# B&R Automation Studio project pneutrunk_plc (part 2)

#### regulator_FF_PI.c
```c
/*
 * regulator_FF_PI.c
 *
 * Academic License - for use in teaching, academic research, and meeting
 * course requirements at degree granting institutions only.  Not for
 * government, commercial, or other organizational use.
 *
 * Code generation for model "regulator_FF_PI".
 *
 * Model version              : 1.96
 * Simulink Coder version : 9.6 (R2021b) 14-May-2021
 * C source code generated on : Tue Apr  5 15:19:23 2022
 *
 * Target selection: bur_grt.tlc
 * Note: GRT includes extra infrastructure and instrumentation for prototyping
 * Embedded hardware selection: Intel->x86/Pentium
 * Code generation objectives: Unspecified
 * Validation result: Not run
 */

#include "regulator_FF_PI.h"
#include "regulator_FF_PI_private.h"

/* Forward declaration for local functions */
static real32_T regulator_FF_PI_norm(const real32_T x[4], struct FF_PID* inst);

/* Function for MATLAB Function: '<S5>/requested alfa 2 deltaz1' */
static real32_T regulator_FF_PI_norm(const real32_T x[4], struct FF_PID* inst)
{
  real32_T absxk;
  real32_T scale;
  real32_T t;
  real32_T y;
  scale = 1.29246971E-26F;
  absxk = fabsf(x[0]);
  if (absxk > 1.29246971E-26F) {
    y = 1.0F;
    scale = absxk;
  } else {
    t = absxk / 1.29246971E-26F;
    y = t * t;
  }

  absxk = fabsf(x[1]);
  if (absxk > scale) {
    t = scale / absxk;
    y = y * t * t + 1.0F;
    scale = absxk;
  } else {
    t = absxk / scale;
    y += t * t;
  }

  absxk = fabsf(x[2]);
  if (absxk > scale) {
    t = scale / absxk;
    y = y * t * t + 1.0F;
    scale = absxk;
  } else {
    t = absxk / scale;
    y += t * t;
  }

  absxk = fabsf(x[3]);
  if (absxk > scale) {
    t = scale / absxk;
    y = y * t * t + 1.0F;
    scale = absxk;
  } else {
    t = absxk / scale;
    y += t * t;
  }

  return scale * sqrtf(y);
}

/* Model step function */
void regulator_FF_PI_step(RT_MODEL_regulator_FF_PI_T *const regulator_FF_PI_M, struct FF_PID* inst)
{
  B_regulator_FF_PI_T *regulator_FF_PI_B = regulator_FF_PI_M->blockIO;
  DW_regulator_FF_PI_T *regulator_FF_PI_DW = regulator_FF_PI_M->dwork;
  real_T oblast_bodov[114];
  real_T Tz23[16];
  real_T Blue0_tmp[4];
  real_T Yellow0_tmp[4];
  real_T A1;
  real_T A2;
  real_T rtb_out;
  real_T tlaky_idx_0;
  real_T tlaky_idx_1;
  real_T tlaky_idx_2;
  real_T tmp;
  real_T tolerancia_bodov;
  real_T tolerancia_tlakov;
  int32_T Tz23_tmp;
  int32_T counter3;
  int32_T i;
  int32_T k;
  real32_T rtb_MultiportSwitch[114];
  real32_T rozdiel[95];
  real32_T vzd_bodov[76];
  real32_T AlphaY_0[16];
  real32_T HTransform[16];
  real32_T HTransform_tmp_1[16];
  real32_T Tz23_0[16];
  real32_T Blue0_tmp_0[4];
  real32_T Green0_tmp_tmp_0[4];
  real32_T Yellow0_tmp_0[4];
  real32_T Yellow0_tmp_1[4];
  real32_T AlphaX;
  real32_T AlphaY;
  real32_T akt_u_idx_2;
  real32_T akt_u_idx_3;
  real32_T akt_u_idx_4;
  real32_T rozdiel_tmp;
  real32_T vzd_bodov_tmp;
  int8_T Green0_tmp_tmp[4];
  int8_T HTransform_tmp[4];
  int8_T HTransform_tmp_0[4];

  /* S-Function (bur_in): '<Root>/Input1' */
  regulator_FF_PI_B->Input1 = inst->ref_alfa_x;

  /* S-Function (bur_in): '<Root>/Input2' */
  regulator_FF_PI_B->Input2 = inst->ref_alfa_y;

  /* S-Function (bur_in): '<Root>/Input3' */
  regulator_FF_PI_B->Input3 = inst->real_alfa_x;

  /* S-Function (bur_in): '<Root>/Input4' */
  regulator_FF_PI_B->Input4 = inst->real_alfa_y;

  /* MATLAB Function: '<S5>/requested alfa 2 deltaz1' incorporates:
   *  Constant: '<S5>/Constant1'
   */
  AlphaX = regulator_FF_PI_B->Input1 * 3.14159274F / 180.0F;
  AlphaY = -regulator_FF_PI_B->Input2 * 3.14159274F / 180.0F;
  Tz23[2] = 0.0;
  Tz23[6] = 0.0;
  Tz23[10] = 1.0;
  Tz23[14] = 57.5;
  akt_u_idx_2 = sinf(AlphaY);
  AlphaY = cosf(AlphaY);
  akt_u_idx_3 = sinf(AlphaX);
  AlphaX = cosf(AlphaX);
  AlphaY_0[0] = AlphaY;
  AlphaY_0[4] = 0.0F;
  AlphaY_0[8] = akt_u_idx_2;
  AlphaY_0[12] = 0.0F;
  AlphaY_0[2] = -akt_u_idx_2;
  AlphaY_0[6] = 0.0F;
  AlphaY_0[10] = AlphaY;
  AlphaY_0[14] = 0.0F;
  Tz23[0] = 1.0;
  Tz23[1] = 0.0;
  Tz23[3] = 0.0;
  HTransform_tmp_0[0] = 1;
  AlphaY_0[1] = 0.0F;
  AlphaY_0[3] = 0.0F;
  HTransform_tmp[0] = 0;
  Tz23[4] = 0.0;
  Tz23[5] = 1.0;
  Tz23[7] = 0.0;
  HTransform_tmp_0[1] = 0;
  AlphaY_0[5] = 1.0F;
  AlphaY_0[7] = 0.0F;
  HTransform_tmp[1] = 0;
  Tz23[8] = 0.0;
  Tz23[9] = 0.0;
  Tz23[11] = 0.0;
  HTransform_tmp_0[2] = 0;
  AlphaY_0[9] = 0.0F;
  AlphaY_0[11] = 0.0F;
  HTransform_tmp[2] = 0;
  Tz23[12] = 0.0;
  Tz23[13] = 0.0;
  Tz23[15] = 1.0;
  HTransform_tmp_0[3] = 0;
  AlphaY_0[13] = 0.0F;
  AlphaY_0[15] = 1.0F;
  HTransform_tmp[3] = 1;
  HTransform_tmp_1[1] = 0.0F;
  HTransform_tmp_1[5] = AlphaX;
  HTransform_tmp_1[9] = -akt_u_idx_3;
  HTransform_tmp_1[13] = 0.0F;
  HTransform_tmp_1[2] = 0.0F;
  HTransform_tmp_1[6] = akt_u_idx_3;
  HTransform_tmp_1[10] = AlphaX;
  HTransform_tmp_1[14] = 0.0F;
  for (i = 0; i < 4; i++) {
    for (k = 0; k < 4; k++) {
      counter3 = k << 2;
      Tz23_tmp = i + counter3;
      Tz23_0[Tz23_tmp] = 0.0F;
      Tz23_0[Tz23_tmp] += AlphaY_0[counter3] * (real32_T)Tz23[i];
      Tz23_0[Tz23_tmp] += AlphaY_0[counter3 + 1] * (real32_T)Tz23[i + 4];
      Tz23_0[Tz23_tmp] += AlphaY_0[counter3 + 2] * (real32_T)Tz23[i + 8];
      Tz23_0[Tz23_tmp] += AlphaY_0[counter3 + 3] * (real32_T)Tz23[i + 12];
    }

    counter3 = i << 2;
    HTransform_tmp_1[counter3] = HTransform_tmp_0[i];
    HTransform_tmp_1[counter3 + 3] = HTransform_tmp[i];
  }

  Green0_tmp_tmp[0] = 85;
  Green0_tmp_tmp[1] = 0;
  Green0_tmp_tmp[2] = 0;
  Green0_tmp_tmp[3] = 1;
  Yellow0_tmp[0] = -42.5;
  Yellow0_tmp[1] = 73.612159321677282;
  Yellow0_tmp[2] = 0.0;
  Yellow0_tmp[3] = 1.0;
  Blue0_tmp[0] = -42.5;
  Blue0_tmp[1] = -73.612159321677282;
  Blue0_tmp[2] = 0.0;
  Blue0_tmp[3] = 1.0;
  for (i = 0; i < 4; i++) {
    for (k = 0; k < 4; k++) {
      counter3 = k << 2;
      Tz23_tmp = i + counter3;
      AlphaY_0[Tz23_tmp] = 0.0F;
      AlphaY_0[Tz23_tmp] += HTransform_tmp_1[counter3] * Tz23_0[i];
      AlphaY_0[Tz23_tmp] += HTransform_tmp_1[counter3 + 1] * Tz23_0[i + 4];
      AlphaY_0[Tz23_tmp] += HTransform_tmp_1[counter3 + 2] * Tz23_0[i + 8];
      AlphaY_0[Tz23_tmp] += HTransform_tmp_1[counter3 + 3] * Tz23_0[i + 12];
    }

    akt_u_idx_2 = 0.0F;
    akt_u_idx_3 = 0.0F;
    akt_u_idx_4 = 0.0F;
    for (k = 0; k < 4; k++) {
      counter3 = k << 2;
      Tz23_tmp = i + counter3;
      HTransform[Tz23_tmp] = 0.0F;
      HTransform[Tz23_tmp] += (real32_T)Tz23[counter3] * AlphaY_0[i];
      HTransform[Tz23_tmp] += (real32_T)Tz23[counter3 + 1] * AlphaY_0[i + 4];
      HTransform[Tz23_tmp] += (real32_T)Tz23[counter3 + 2] * AlphaY_0[i + 8];
      HTransform[Tz23_tmp] += (real32_T)Tz23[counter3 + 3] * AlphaY_0[i + 12];
      akt_u_idx_2 += HTransform[Tz23_tmp] * (real32_T)Green0_tmp_tmp[k];
      akt_u_idx_3 += HTransform[Tz23_tmp] * (real32_T)Yellow0_tmp[k];
      akt_u_idx_4 += HTransform[Tz23_tmp] * (real32_T)Blue0_tmp[k];
    }

    Green0_tmp_tmp_0[i] = (real32_T)Green0_tmp_tmp[i] - akt_u_idx_2;
    Yellow0_tmp_0[i] = (real32_T)Yellow0_tmp[i] - akt_u_idx_3;
    Blue0_tmp_0[i] = (real32_T)Blue0_tmp[i] - akt_u_idx_4;
  }

  AlphaX = regulator_FF_PI_B->Input3 * 3.14159274F / 180.0F;
  AlphaY = -regulator_FF_PI_B->Input4 * 3.14159274F / 180.0F;
  akt_u_idx_2 = sinf(AlphaY);
  AlphaY = cosf(AlphaY);
  akt_u_idx_3 = sinf(AlphaX);
  AlphaX = cosf(AlphaX);
  AlphaY_0[0] = AlphaY;
  AlphaY_0[4] = 0.0F;
  AlphaY_0[8] = akt_u_idx_2;
  AlphaY_0[12] = 0.0F;
  AlphaY_0[2] = -akt_u_idx_2;
  AlphaY_0[6] = 0.0F;
  AlphaY_0[10] = AlphaY;
  AlphaY_0[14] = 0.0F;
  AlphaY_0[1] = 0.0F;
  AlphaY_0[3] = 0.0F;
  AlphaY_0[5] = 1.0F;
  AlphaY_0[7] = 0.0F;
  AlphaY_0[9] = 0.0F;
  AlphaY_0[11] = 0.0F;
  AlphaY_0[13] = 0.0F;
  AlphaY_0[15] = 1.0F;
  HTransform_tmp_1[1] = 0.0F;
  HTransform_tmp_1[5] = AlphaX;
  HTransform_tmp_1[9] = -akt_u_idx_3;
  HTransform_tmp_1[13] = 0.0F;
  HTransform_tmp_1[2] = 0.0F;
  HTransform_tmp_1[6] = akt_u_idx_3;
  HTransform_tmp_1[10] = AlphaX;
  HTransform_tmp_1[14] = 0.0F;
  for (i = 0; i < 4; i++) {
    for (k = 0; k < 4; k++) {
      counter3 = k << 2;
      Tz23_tmp = i + counter3;
      Tz23_0[Tz23_tmp] = 0.0F;
      Tz23_0[Tz23_tmp] += AlphaY_0[counter3] * (real32_T)Tz23[i];
      Tz23_0[Tz23_tmp] += AlphaY_0[counter3 + 1] * (real32_T)Tz23[i + 4];
      Tz23_0[Tz23_tmp] += AlphaY_0[counter3 + 2] * (real32_T)Tz23[i + 8];
      Tz23_0[Tz23_tmp] += AlphaY_0[counter3 + 3] * (real32_T)Tz23[i + 12];
    }

    counter3 = i << 2;
    HTransform_tmp_1[counter3] = HTransform_tmp_0[i];
    HTransform_tmp_1[counter3 + 3] = HTransform_tmp[i];
  }

  Yellow0_tmp[0] = -42.5;
  Yellow0_tmp[1] = 73.612159321677282;
  Yellow0_tmp[2] = 0.0;
  Yellow0_tmp[3] = 1.0;
  Blue0_tmp[0] = -42.5;
  Blue0_tmp[1] = -73.612159321677282;
  Blue0_tmp[2] = 0.0;
  Blue0_tmp[3] = 1.0;
  for (i = 0; i < 4; i++) {
    for (k = 0; k < 4; k++) {
      counter3 = k << 2;
      Tz23_tmp = i + counter3;
      AlphaY_0[Tz23_tmp] = 0.0F;
      AlphaY_0[Tz23_tmp] += HTransform_tmp_1[counter3] * Tz23_0[i];
      AlphaY_0[Tz23_tmp] += HTransform_tmp_1[counter3 + 1] * Tz23_0[i + 4];
      AlphaY_0[Tz23_tmp] += HTransform_tmp_1[counter3 + 2] * Tz23_0[i + 8];
      AlphaY_0[Tz23_tmp] += HTransform_tmp_1[counter3 + 3] * Tz23_0[i + 12];
    }

    akt_u_idx_2 = 0.0F;
    for (k = 0; k < 4; k++) {
      counter3 = k << 2;
      Tz23_tmp = i + counter3;
      HTransform[Tz23_tmp] = 0.0F;
      HTransform[Tz23_tmp] += (real32_T)Tz23[counter3] * AlphaY_0[i];
      HTransform[Tz23_tmp] += (real32_T)Tz23[counter3 + 1] * AlphaY_0[i + 4];
      HTransform[Tz23_tmp] += (real32_T)Tz23[counter3 + 2] * AlphaY_0[i + 8];
      HTransform[Tz23_tmp] += (real32_T)Tz23[counter3 + 3] * AlphaY_0[i + 12];
      akt_u_idx_2 += HTransform[Tz23_tmp] * (real32_T)Yellow0_tmp[k];
    }

    Yellow0_tmp_1[i] = (real32_T)Yellow0_tmp[i] - akt_u_idx_2;
  }

  /* Sum: '<S2>/Sum' incorporates:
   *  Constant: '<S11>/cylinder height'
   *  Constant: '<S9>/cylinder height'
   *  Gain: '<S5>/Gain'
   *  Gain: '<S5>/Gain3'
   *  MATLAB Function: '<S5>/requested alfa 2 deltaz1'
   *  Sum: '<S11>/Sum'
   *  Sum: '<S9>/Sum'
   */
  A2 = (0.001F * regulator_FF_PI_norm(Yellow0_tmp_1, inst) - 0.115) - (0.001F *
    regulator_FF_PI_norm(Yellow0_tmp_0, inst) - 0.115);

  /* S-Function (bur_in): '<Root>/Input11' */
  regulator_FF_PI_B->Input11 = inst->P_parameter;

  /* S-Function (bur_in): '<Root>/Input5' */
  regulator_FF_PI_B->Input5 = inst->reset_PID_blue;

  /* DiscreteIntegrator: '<S143>/Integrator' */
  if ((regulator_FF_PI_B->Input5 <= 0.0F) &&
      (regulator_FF_PI_DW->Integrator_PrevResetState == 1)) {
    regulator_FF_PI_DW->Integrator_DSTATE = 0.0;
  }

  /* S-Function (bur_in): '<Root>/Input13' */
  regulator_FF_PI_B->Input13 = inst->D_parameter;

  /* DiscreteIntegrator: '<S138>/Filter' */
  if ((regulator_FF_PI_B->Input5 <= 0.0F) &&
      (regulator_FF_PI_DW->Filter_PrevResetState == 1)) {
    regulator_FF_PI_DW->Filter_DSTATE = 0.0;
  }

  /* S-Function (bur_in): '<Root>/Input14' */
  regulator_FF_PI_B->Input14 = inst->N_parameter;

  /* Product: '<S146>/NProd Out' incorporates:
   *  DiscreteIntegrator: '<S138>/Filter'
   *  Product: '<S137>/DProd Out'
   *  Sum: '<S138>/SumD'
   */
  A1 = (A2 * regulator_FF_PI_B->Input13 - regulator_FF_PI_DW->Filter_DSTATE) *
    regulator_FF_PI_B->Input14;

  /* S-Function (bur_in): '<Root>/Input8' */
  regulator_FF_PI_B->Input8 = inst->tlak1;

  /* S-Function (bur_in): '<Root>/Input9' */
  regulator_FF_PI_B->Input9 = inst->tlak2;

  /* S-Function (bur_in): '<Root>/Input10' */
  regulator_FF_PI_B->Input10 = inst->tlak3;

  /* MATLAB Function: '<S1>/prepinac' */
  rtb_out = 1.0;
  if ((regulator_FF_PI_B->Input1 < 0.0F) && (regulator_FF_PI_B->Input2 > 0.0F))
  {
    rtb_out = 2.0;
  }

  if ((regulator_FF_PI_B->Input1 > 0.0F) && (regulator_FF_PI_B->Input2 < 0.0F))
  {
    rtb_out = 3.0;
  }

  if ((regulator_FF_PI_B->Input1 <= 0.0F) && (regulator_FF_PI_B->Input2 <= 0.0F))
  {
    rtb_out = 4.0;
  }

  /* End of MATLAB Function: '<S1>/prepinac' */

  /* MultiPortSwitch: '<S1>/Multiport Switch' incorporates:
   *  Constant: '<S1>/Constant'
   *  Constant: '<S1>/Constant1'
   *  Constant: '<S1>/Constant2'
   *  Constant: '<S1>/Constant3'
   */
  switch ((int32_T)rtb_out) {
   case 1:
    for (i = 0; i < 114; i++) {
      rtb_MultiportSwitch[i] = regulator_FF_PI_ConstP.Constant_Value_m[i];
    }
    break;

   case 2:
    for (i = 0; i < 114; i++) {
      rtb_MultiportSwitch[i] = regulator_FF_PI_ConstP.Constant1_Value_b[i];
    }
    break;

   case 3:
    for (i = 0; i < 114; i++) {
      rtb_MultiportSwitch[i] = regulator_FF_PI_ConstP.Constant3_Value[i];
    }
    break;

   default:
    for (i = 0; i < 114; i++) {
      rtb_MultiportSwitch[i] = regulator_FF_PI_ConstP.Constant2_Value[i];
    }
    break;
  }

  /* End of MultiPortSwitch: '<S1>/Multiport Switch' */

  /* MATLAB Function: '<S1>/ff' incorporates:
   *  MultiPortSwitch: '<S1>/Multiport Switch'
   */
  akt_u_idx_2 = regulator_FF_PI_B->Input8;
  akt_u_idx_3 = regulator_FF_PI_B->Input9;
  akt_u_idx_4 = regulator_FF_PI_B->Input10;
  tolerancia_bodov = 2.0;
  tolerancia_tlakov = 2.0;
  counter3 = 0;
  tlaky_idx_0 = 0.0;
  tlaky_idx_1 = 0.0;
  tlaky_idx_2 = 0.0;
  for (k = 0; k < 19; k++) {
    rozdiel[k] = rtb_MultiportSwitch[k] - regulator_FF_PI_B->Input1;
    rozdiel[k + 19] = rtb_MultiportSwitch[k + 19] - regulator_FF_PI_B->Input2;
    AlphaX = rtb_MultiportSwitch[k + 38];
    rozdiel[k + 38] = AlphaX;
    AlphaY = rtb_MultiportSwitch[k + 57];
    rozdiel[k + 57] = AlphaY;
    rozdiel_tmp = rtb_MultiportSwitch[k + 76];
    rozdiel[k + 76] = rozdiel_tmp;
    vzd_bodov_tmp = rozdiel[k + 19];
    vzd_bodov[k] = sqrtf(vzd_bodov_tmp * vzd_bodov_tmp + rozdiel[k] * rozdiel[k]);
    vzd_bodov[k + 19] = AlphaX;
    vzd_bodov[k + 38] = AlphaY;
    vzd_bodov[k + 57] = rozdiel_tmp;
  }

  for (i = 0; i < 114; i++) {
    oblast_bodov[i] = 0.0;
  }

  rtb_out = 0.0;
  if (regulator_FF_PI_B->Input8 <= 2.0F) {
    akt_u_idx_2 = 2.0F;
  }

  if (regulator_FF_PI_B->Input9 <= 2.0F) {
    akt_u_idx_3 = 2.0F;
  }

  if (regulator_FF_PI_B->Input10 <= 2.0F) {
    akt_u_idx_4 = 2.0F;
  }

  int32_T exitg1;
  do {
    exitg1 = 0;
    for (k = 0; k < 19; k++) {
      if ((vzd_bodov[k] <= tolerancia_bodov) && (fabsf(((akt_u_idx_2 +
              akt_u_idx_3) + akt_u_idx_4) - rtb_MultiportSwitch[k + 95]) <=
           tolerancia_tlakov)) {
        rtb_out++;
        for (i = 0; i < 6; i++) {
          oblast_bodov[((int32_T)rtb_out + 19 * i) - 1] = rtb_MultiportSwitch[19
            * i + k];
        }

        rozdiel_tmp = (real32_T)oblast_bodov[(int32_T)rtb_out - 1] -
          regulator_FF_PI_B->Input1;
        vzd_bodov_tmp = (real32_T)oblast_bodov[(int32_T)rtb_out + 18] -
          regulator_FF_PI_B->Input2;
        rozdiel_tmp = sqrtf(rozdiel_tmp * rozdiel_tmp + vzd_bodov_tmp *
                            vzd_bodov_tmp);
        if (rozdiel_tmp <= 0.5F) {
          if (counter3 == 0) {
            counter3 = 1;
            tlaky_idx_0 = oblast_bodov[(int32_T)rtb_out + 37];
            tlaky_idx_1 = oblast_bodov[(int32_T)rtb_out + 56];
            tlaky_idx_2 = oblast_bodov[(int32_T)rtb_out + 75];
          } else {
            AlphaX = (real32_T)oblast_bodov[(int32_T)(rtb_out - 1.0) - 1] -
              regulator_FF_PI_B->Input1;
            AlphaY = (real32_T)oblast_bodov[(int32_T)(rtb_out - 1.0) + 18] -
              regulator_FF_PI_B->Input2;
            if (rozdiel_tmp < sqrtf(AlphaX * AlphaX + AlphaY * AlphaY)) {
              tlaky_idx_0 = oblast_bodov[(int32_T)rtb_out + 37];
              tlaky_idx_1 = oblast_bodov[(int32_T)rtb_out + 56];
              tlaky_idx_2 = oblast_bodov[(int32_T)rtb_out + 75];
            }
          }
        }
      }
    }

    if (rtb_out == 0.0) {
      tolerancia_bodov++;
      tolerancia_tlakov++;
    } else {
      exitg1 = 1;
    }
  } while (exitg1 == 0);

  if (counter3 == 0) {
    tolerancia_bodov = oblast_bodov[38];
    for (counter3 = 2; counter3 <= (int32_T)rtb_out; counter3++) {
      tolerancia_bodov += oblast_bodov[counter3 + 37];
    }

    tolerancia_tlakov = oblast_bodov[57];
    for (counter3 = 2; counter3 <= (int32_T)rtb_out; counter3++) {
      tolerancia_tlakov += oblast_bodov[counter3 + 56];
    }

    tlaky_idx_2 = oblast_bodov[76];
    for (counter3 = 2; counter3 <= (int32_T)rtb_out; counter3++) {
      tlaky_idx_2 += oblast_bodov[counter3 + 75];
    }

    tlaky_idx_0 = tolerancia_bodov / (real_T)(int32_T)rtb_out;
    tlaky_idx_1 = tolerancia_tlakov / (real_T)(int32_T)rtb_out;
    tlaky_idx_2 /= (real_T)(int32_T)rtb_out;
  }

  /* Switch: '<Root>/Switch2' incorporates:
   *  DiscreteIntegrator: '<S143>/Integrator'
   *  Product: '<S148>/PProd Out'
   *  Sum: '<S152>/Sum'
   */
  if (regulator_FF_PI_B->Input5 > 0.0F) {
    tmp = (A2 * regulator_FF_PI_B->Input11 +
           regulator_FF_PI_DW->Integrator_DSTATE) + A1;
  } else {
    tmp = 0.0;
  }

  /* End of Switch: '<Root>/Switch2' */

  /* Sum: '<Root>/Sum' incorporates:
   *  MATLAB Function: '<S1>/ff'
   */
  regulator_FF_PI_B->Sum = (real32_T)(tmp + tlaky_idx_0);

  /* S-Function (bur_out): '<Root>/Output1' */
  inst->Blue_tab = regulator_FF_PI_B->Sum;

  /* MATLAB Function: '<S5>/requested alfa 2 deltaz1' */
  for (i = 0; i < 4; i++) {
    Yellow0_tmp_0[i] = (real32_T)Green0_tmp_tmp[i] - (HTransform[i] * 85.0F +
      HTransform[i + 12]);
  }

  /* Sum: '<S2>/Sum2' incorporates:
   *  Constant: '<S12>/cylinder height'
   *  Constant: '<S14>/cylinder height'
   *  Gain: '<S5>/Gain1'
   *  Gain: '<S5>/Gain4'
   *  MATLAB Function: '<S5>/requested alfa 2 deltaz1'
   *  Sum: '<S12>/Sum'
   *  Sum: '<S14>/Sum'
   */
  tolerancia_tlakov = (0.001F * regulator_FF_PI_norm(Yellow0_tmp_0, inst) - 0.115) -
    (0.001F * regulator_FF_PI_norm(Green0_tmp_tmp_0, inst) - 0.115);

  /* S-Function (bur_in): '<Root>/Input7' */
  regulator_FF_PI_B->Input7 = inst->reset_PID_green;

  /* DiscreteIntegrator: '<S95>/Integrator' */
  if ((regulator_FF_PI_B->Input7 <= 0.0F) &&
      (regulator_FF_PI_DW->Integrator_PrevResetState_l == 1)) {
    regulator_FF_PI_DW->Integrator_DSTATE_o = 0.0;
  }

  /* DiscreteIntegrator: '<S90>/Filter' */
  if ((regulator_FF_PI_B->Input7 <= 0.0F) &&
      (regulator_FF_PI_DW->Filter_PrevResetState_e == 1)) {
    regulator_FF_PI_DW->Filter_DSTATE_f = 0.0;
  }

  /* Product: '<S98>/NProd Out' incorporates:
   *  DiscreteIntegrator: '<S90>/Filter'
   *  Product: '<S89>/DProd Out'
   *  Sum: '<S90>/SumD'
   */
  rtb_out = (tolerancia_tlakov * regulator_FF_PI_B->Input13 -
             regulator_FF_PI_DW->Filter_DSTATE_f) * regulator_FF_PI_B->Input14;

  /* Switch: '<Root>/Switch' incorporates:
   *  DiscreteIntegrator: '<S95>/Integrator'
   *  Product: '<S100>/PProd Out'
   *  Sum: '<S104>/Sum'
   */
  if (regulator_FF_PI_B->Input7 > 0.0F) {
    tmp = (tolerancia_tlakov * regulator_FF_PI_B->Input11 +
           regulator_FF_PI_DW->Integrator_DSTATE_o) + rtb_out;
  } else {
    tmp = 0.0;
  }

  /* End of Switch: '<Root>/Switch' */

  /* Sum: '<Root>/Sum2' incorporates:
   *  MATLAB Function: '<S1>/ff'
   */
  regulator_FF_PI_B->Sum2 = (real32_T)(tmp + tlaky_idx_2);

  /* S-Function (bur_out): '<Root>/Output2' */
  inst->Yellow_tab = regulator_FF_PI_B->Sum2;

  /* MATLAB Function: '<S5>/requested alfa 2 deltaz1' */
  for (i = 0; i < 4; i++) {
    Green0_tmp_tmp_0[i] = (real32_T)Blue0_tmp[i] - ((HTransform[i + 4] *
      -73.6121597F + HTransform[i] * -42.5F) + HTransform[i + 12]);
  }

  /* Sum: '<S2>/Sum1' incorporates:
   *  Constant: '<S10>/cylinder height'
   *  Constant: '<S13>/cylinder height'
   *  Gain: '<S5>/Gain2'
   *  Gain: '<S5>/Gain5'
   *  MATLAB Function: '<S5>/requested alfa 2 deltaz1'
   *  Sum: '<S10>/Sum'
   *  Sum: '<S13>/Sum'
   */
  tlaky_idx_2 = (0.001F * regulator_FF_PI_norm(Green0_tmp_tmp_0, inst) - 0.115) -
    (0.001F * regulator_FF_PI_norm(Blue0_tmp_0, inst) - 0.115);

  /* S-Function (bur_in): '<Root>/Input6' */
  regulator_FF_PI_B->Input6 = inst->reset_PID_yellow;

  /* DiscreteIntegrator: '<S47>/Integrator' */
  if ((regulator_FF_PI_B->Input6 <= 0.0F) &&
      (regulator_FF_PI_DW->Integrator_PrevResetState_e == 1)) {
    regulator_FF_PI_DW->Integrator_DSTATE_i = 0.0;
  }

  /* DiscreteIntegrator: '<S42>/Filter' */
  if ((regulator_FF_PI_B->Input6 <= 0.0F) &&
      (regulator_FF_PI_DW->Filter_PrevResetState_h == 1)) {
    regulator_FF_PI_DW->Filter_DSTATE_a = 0.0;
  }

  /* Product: '<S50>/NProd Out' incorporates:
   *  DiscreteIntegrator: '<S42>/Filter'
   *  Product: '<S41>/DProd Out'
   *  Sum: '<S42>/SumD'
   */
  tolerancia_bodov = (tlaky_idx_2 * regulator_FF_PI_B->Input13 -
                      regulator_FF_PI_DW->Filter_DSTATE_a) *
    regulator_FF_PI_B->Input14;

  /* Switch: '<Root>/Switch1' incorporates:
   *  DiscreteIntegrator: '<S47>/Integrator'
   *  Product: '<S52>/PProd Out'
   *  Sum: '<S56>/Sum'
   */
  if (regulator_FF_PI_B->Input6 > 0.0F) {
    tmp = (tlaky_idx_2 * regulator_FF_PI_B->Input11 +
           regulator_FF_PI_DW->Integrator_DSTATE_i) + tolerancia_bodov;
  } else {
    tmp = 0.0;
  }

  /* End of Switch: '<Root>/Switch1' */

  /* Sum: '<Root>/Sum1' incorporates:
   *  MATLAB Function: '<S1>/ff'
   */
  regulator_FF_PI_B->Sum1 = (real32_T)(tmp + tlaky_idx_1);

  /* S-Function (bur_out): '<Root>/Output4' */
  inst->Green_tab = regulator_FF_PI_B->Sum1;

  /* S-Function (bur_in): '<Root>/Input12' */
  regulator_FF_PI_B->Input12 = inst->I_parameter;

  /* Product: '<S44>/IProd Out' */
  tlaky_idx_0 = tlaky_idx_2 * regulator_FF_PI_B->Input12;

  /* Product: '<S92>/IProd Out' */
  tolerancia_tlakov *= regulator_FF_PI_B->Input12;

  /* Product: '<S140>/IProd Out' */
  A2 *= regulator_FF_PI_B->Input12;

  /* Update for DiscreteIntegrator: '<S143>/Integrator' */
  regulator_FF_PI_DW->Integrator_DSTATE += 0.002 * A2;
  if (regulator_FF_PI_B->Input5 > 0.0F) {
    regulator_FF_PI_DW->Integrator_PrevResetState = 1;
  } else if (regulator_FF_PI_B->Input5 < 0.0F) {
    regulator_FF_PI_DW->Integrator_PrevResetState = -1;
  } else if (regulator_FF_PI_B->Input5 == 0.0F) {
    regulator_FF_PI_DW->Integrator_PrevResetState = 0;
  } else {
    regulator_FF_PI_DW->Integrator_PrevResetState = 2;
  }

  /* End of Update for DiscreteIntegrator: '<S143>/Integrator' */

  /* Update for DiscreteIntegrator: '<S138>/Filter' */
  regulator_FF_PI_DW->Filter_DSTATE += 0.002 * A1;
  if (regulator_FF_PI_B->Input5 > 0.0F) {
    regulator_FF_PI_DW->Filter_PrevResetState = 1;
  } else if (regulator_FF_PI_B->Input5 < 0.0F) {
    regulator_FF_PI_DW->Filter_PrevResetState = -1;
  } else if (regulator_FF_PI_B->Input5 == 0.0F) {
    regulator_FF_PI_DW->Filter_PrevResetState = 0;
  } else {
    regulator_FF_PI_DW->Filter_PrevResetState = 2;
  }

  /* End of Update for DiscreteIntegrator: '<S138>/Filter' */

  /* Update for DiscreteIntegrator: '<S95>/Integrator' */
  regulator_FF_PI_DW->Integrator_DSTATE_o += 0.002 * tolerancia_tlakov;
  if (regulator_FF_PI_B->Input7 > 0.0F) {
    regulator_FF_PI_DW->Integrator_PrevResetState_l = 1;
  } else if (regulator_FF_PI_B->Input7 < 0.0F) {
    regulator_FF_PI_DW->Integrator_PrevResetState_l = -1;
  } else if (regulator_FF_PI_B->Input7 == 0.0F) {
    regulator_FF_PI_DW->Integrator_PrevResetState_l = 0;
  } else {
    regulator_FF_PI_DW->Integrator_PrevResetState_l = 2;
  }

  /* End of Update for DiscreteIntegrator: '<S95>/Integrator' */

  /* Update for DiscreteIntegrator: '<S90>/Filter' */
  regulator_FF_PI_DW->Filter_DSTATE_f += 0.002 * rtb_out;
  if (regulator_FF_PI_B->Input7 > 0.0F) {
    regulator_FF_PI_DW->Filter_PrevResetState_e = 1;
  } else if (regulator_FF_PI_B->Input7 < 0.0F) {
    regulator_FF_PI_DW->Filter_PrevResetState_e = -1;
  } else if (regulator_FF_PI_B->Input7 == 0.0F) {
    regulator_FF_PI_DW->Filter_PrevResetState_e = 0;
  } else {
    regulator_FF_PI_DW->Filter_PrevResetState_e = 2;
  }

  /* End of Update for DiscreteIntegrator: '<S90>/Filter' */

  /* Update for DiscreteIntegrator: '<S47>/Integrator' */
  regulator_FF_PI_DW->Integrator_DSTATE_i += 0.002 * tlaky_idx_0;
  if (regulator_FF_PI_B->Input6 > 0.0F) {
    regulator_FF_PI_DW->Integrator_PrevResetState_e = 1;
  } else if (regulator_FF_PI_B->Input6 < 0.0F) {
    regulator_FF_PI_DW->Integrator_PrevResetState_e = -1;
  } else if (regulator_FF_PI_B->Input6 == 0.0F) {
    regulator_FF_PI_DW->Integrator_PrevResetState_e = 0;
  } else {
    regulator_FF_PI_DW->Integrator_PrevResetState_e = 2;
  }

  /* End of Update for DiscreteIntegrator: '<S47>/Integrator' */

  /* Update for DiscreteIntegrator: '<S42>/Filter' */
  regulator_FF_PI_DW->Filter_DSTATE_a += 0.002 * tolerancia_bodov;
  if (regulator_FF_PI_B->Input6 > 0.0F) {
    regulator_FF_PI_DW->Filter_PrevResetState_h = 1;
  } else if (regulator_FF_PI_B->Input6 < 0.0F) {
    regulator_FF_PI_DW->Filter_PrevResetState_h = -1;
  } else if (regulator_FF_PI_B->Input6 == 0.0F) {
    regulator_FF_PI_DW->Filter_PrevResetState_h = 0;
  } else {
    regulator_FF_PI_DW->Filter_PrevResetState_h = 2;
  }

  /* End of Update for DiscreteIntegrator: '<S42>/Filter' */
}

/* Model initialize function */
void regulator_FF_PI_initialize(RT_MODEL_regulator_FF_PI_T *const
  regulator_FF_PI_M, struct FF_PID* inst)
{
  DW_regulator_FF_PI_T *regulator_FF_PI_DW = regulator_FF_PI_M->dwork;

  /* InitializeConditions for DiscreteIntegrator: '<S143>/Integrator' */
  regulator_FF_PI_DW->Integrator_DSTATE = 0.0;
  regulator_FF_PI_DW->Integrator_PrevResetState = 2;

  /* InitializeConditions for DiscreteIntegrator: '<S138>/Filter' */
  regulator_FF_PI_DW->Filter_DSTATE = 0.0;
  regulator_FF_PI_DW->Filter_PrevResetState = 2;

  /* InitializeConditions for DiscreteIntegrator: '<S95>/Integrator' */
  regulator_FF_PI_DW->Integrator_DSTATE_o = 0.0;
  regulator_FF_PI_DW->Integrator_PrevResetState_l = 2;

  /* InitializeConditions for DiscreteIntegrator: '<S90>/Filter' */
  regulator_FF_PI_DW->Filter_DSTATE_f = 0.0;
  regulator_FF_PI_DW->Filter_PrevResetState_e = 2;

  /* InitializeConditions for DiscreteIntegrator: '<S47>/Integrator' */
  regulator_FF_PI_DW->Integrator_DSTATE_i = 0.0;
  regulator_FF_PI_DW->Integrator_PrevResetState_e = 2;

  /* InitializeConditions for DiscreteIntegrator: '<S42>/Filter' */
  regulator_FF_PI_DW->Filter_DSTATE_a = 0.0;
  regulator_FF_PI_DW->Filter_PrevResetState_h = 2;
}

/* Model terminate function */
void regulator_FF_PI_terminate(RT_MODEL_regulator_FF_PI_T * regulator_FF_PI_M, struct FF_PID* inst)
{}

/* Model data allocation function */
void regulator_FF_PI_initializeMemory(RT_MODEL_regulator_FF_PI_T* const regulator_FF_PI_M, struct FF_PID * inst)
{  /* states (dwork) */
  {
  }

  {
    B_regulator_FF_PI_T *regulator_FF_PI_B = regulator_FF_PI_M->blockIO;
    DW_regulator_FF_PI_T *regulator_FF_PI_DW = regulator_FF_PI_M->dwork;

    /* block I/O */
    {
      regulator_FF_PI_B->Input1 = 0.0F;
      regulator_FF_PI_B->Input2 = 0.0F;
      regulator_FF_PI_B->Input3 = 0.0F;
      regulator_FF_PI_B->Input4 = 0.0F;
      regulator_FF_PI_B->Input11 = 0.0F;
      regulator_FF_PI_B->Input5 = 0.0F;
      regulator_FF_PI_B->Input13 = 0.0F;
      regulator_FF_PI_B->Input14 = 0.0F;
      regulator_FF_PI_B->Input8 = 0.0F;
      regulator_FF_PI_B->Input9 = 0.0F;
      regulator_FF_PI_B->Input10 = 0.0F;
      regulator_FF_PI_B->Sum = 0.0F;
      regulator_FF_PI_B->Input7 = 0.0F;
      regulator_FF_PI_B->Sum2 = 0.0F;
      regulator_FF_PI_B->Input6 = 0.0F;
      regulator_FF_PI_B->Sum1 = 0.0F;
      regulator_FF_PI_B->Input12 = 0.0F;
    }

    /* states (dwork) */
    (void) memset((void *)regulator_FF_PI_DW, 0,
                  sizeof(DW_regulator_FF_PI_T));
    regulator_FF_PI_DW->Integrator_DSTATE = 0.0;
    regulator_FF_PI_DW->Filter_DSTATE = 0.0;
    regulator_FF_PI_DW->Integrator_DSTATE_o = 0.0;
    regulator_FF_PI_DW->Filter_DSTATE_f = 0.0;
    regulator_FF_PI_DW->Integrator_DSTATE_i = 0.0;
    regulator_FF_PI_DW->Filter_DSTATE_a = 0.0;
  }

}
```

#### regulator_nelin_P.c
```c
/*
 * regulator_nelin_P.c
 *
 * Academic License - for use in teaching, academic research, and meeting
 * course requirements at degree granting institutions only.  Not for
 * government, commercial, or other organizational use.
 *
 * Code generation for model "regulator_nelin_P".
 *
 * Model version              : 1.10
 * Simulink Coder version : 9.6 (R2021b) 14-May-2021
 * C source code generated on : Fri Jul 29 10:48:17 2022
 *
 * Target selection: bur_grt.tlc
 * Note: GRT includes extra infrastructure and instrumentation for prototyping
 * Embedded hardware selection: Intel->x86/Pentium
 * Code generation objectives: Unspecified
 * Validation result: Not run
 */

#include "regulator_nelin_P.h"
#include "regulator_nelin_P_private.h"

/* Forward declaration for local functions */
static real32_T regulator_nelin_P_norm(const real32_T x[4], struct nonL_P* inst);

/* Function for MATLAB Function: '<S1>/requested alfa 2 deltaz1' */
static real32_T regulator_nelin_P_norm(const real32_T x[4], struct nonL_P* inst)
{
  real32_T absxk;
  real32_T scale;
  real32_T t;
  real32_T y;
  scale = 1.29246971E-26F;
  absxk = fabsf(x[0]);
  if (absxk > 1.29246971E-26F) {
    y = 1.0F;
    scale = absxk;
  } else {
    t = absxk / 1.29246971E-26F;
    y = t * t;
  }

  absxk = fabsf(x[1]);
  if (absxk > scale) {
    t = scale / absxk;
    y = y * t * t + 1.0F;
    scale = absxk;
  } else {
    t = absxk / scale;
    y += t * t;
  }

  absxk = fabsf(x[2]);
  if (absxk > scale) {
    t = scale / absxk;
    y = y * t * t + 1.0F;
    scale = absxk;
  } else {
    t = absxk / scale;
    y += t * t;
  }

  absxk = fabsf(x[3]);
  if (absxk > scale) {
    t = scale / absxk;
    y = y * t * t + 1.0F;
    scale = absxk;
  } else {
    t = absxk / scale;
    y += t * t;
  }

  return scale * sqrtf(y);
}

/* Model step function */
void regulator_nelin_P_step(RT_MODEL_regulator_nelin_P_T *const
  regulator_nelin_P_M, struct nonL_P* inst)
{
  B_regulator_nelin_P_T *regulator_nelin_P_B = regulator_nelin_P_M->blockIO;
  real_T Tz23[16];
  real_T Blue0_tmp[4];
  real_T Yellow0_tmp[4];
  int32_T Tz23_tmp;
  int32_T Tz23_tmp_tmp;
  int32_T i;
  int32_T i_0;
  real32_T AlphaY_0[16];
  real32_T HTransform[16];
  real32_T HTransform_tmp_3[16];
  real32_T Tz23_0[16];
  real32_T Blue0_tmp_0[4];
  real32_T Green0_tmp_tmp_0[4];
  real32_T Yellow0_tmp_0[4];
  real32_T Yellow0_tmp_1[4];
  real32_T AlphaX;
  real32_T AlphaY;
  real32_T HTransform_tmp;
  real32_T HTransform_tmp_0;
  int8_T Green0_tmp_tmp[4];
  int8_T HTransform_tmp_1[4];
  int8_T HTransform_tmp_2[4];

  /* S-Function (bur_in): '<Root>/Input1' */
  regulator_nelin_P_B->Input1 = inst->ref_alfa_x;

  /* S-Function (bur_in): '<Root>/Input2' */
  regulator_nelin_P_B->Input2 = inst->ref_alfa_y;

  /* S-Function (bur_in): '<Root>/Input3' */
  regulator_nelin_P_B->Input3 = inst->real_alfa_x;

  /* S-Function (bur_in): '<Root>/Input4' */
  regulator_nelin_P_B->Input4 = inst->real_alfa_y;

  /* MATLAB Function: '<S1>/requested alfa 2 deltaz1' incorporates:
   *  Constant: '<S1>/Constant1'
   */
  AlphaX = regulator_nelin_P_B->Input1 * 3.14159274F / 180.0F;
  AlphaY = -regulator_nelin_P_B->Input2 * 3.14159274F / 180.0F;
  Tz23[2] = 0.0;
  Tz23[6] = 0.0;
  Tz23[10] = 1.0;
  Tz23[14] = 57.5;
  HTransform_tmp = sinf(AlphaY);
  AlphaY = cosf(AlphaY);
  HTransform_tmp_0 = sinf(AlphaX);
  AlphaX = cosf(AlphaX);
  AlphaY_0[0] = AlphaY;
  AlphaY_0[4] = 0.0F;
  AlphaY_0[8] = HTransform_tmp;
  AlphaY_0[12] = 0.0F;
  AlphaY_0[2] = -HTransform_tmp;
  AlphaY_0[6] = 0.0F;
  AlphaY_0[10] = AlphaY;
  AlphaY_0[14] = 0.0F;
  Tz23[0] = 1.0;
  Tz23[1] = 0.0;
  Tz23[3] = 0.0;
  HTransform_tmp_2[0] = 1;
  AlphaY_0[1] = 0.0F;
  AlphaY_0[3] = 0.0F;
  HTransform_tmp_1[0] = 0;
  Tz23[4] = 0.0;
  Tz23[5] = 1.0;
  Tz23[7] = 0.0;
  HTransform_tmp_2[1] = 0;
  AlphaY_0[5] = 1.0F;
  AlphaY_0[7] = 0.0F;
  HTransform_tmp_1[1] = 0;
  Tz23[8] = 0.0;
  Tz23[9] = 0.0;
  Tz23[11] = 0.0;
  HTransform_tmp_2[2] = 0;
  AlphaY_0[9] = 0.0F;
  AlphaY_0[11] = 0.0F;
  HTransform_tmp_1[2] = 0;
  Tz23[12] = 0.0;
  Tz23[13] = 0.0;
  Tz23[15] = 1.0;
  HTransform_tmp_2[3] = 0;
  AlphaY_0[13] = 0.0F;
  AlphaY_0[15] = 1.0F;
  HTransform_tmp_1[3] = 1;
  HTransform_tmp_3[1] = 0.0F;
  HTransform_tmp_3[5] = AlphaX;
  HTransform_tmp_3[9] = -HTransform_tmp_0;
  HTransform_tmp_3[13] = 0.0F;
  HTransform_tmp_3[2] = 0.0F;
  HTransform_tmp_3[6] = HTransform_tmp_0;
  HTransform_tmp_3[10] = AlphaX;
  HTransform_tmp_3[14] = 0.0F;
  for (i = 0; i < 4; i++) {
    for (i_0 = 0; i_0 < 4; i_0++) {
      Tz23_tmp_tmp = i_0 << 2;
      Tz23_tmp = i + Tz23_tmp_tmp;
      Tz23_0[Tz23_tmp] = 0.0F;
      Tz23_0[Tz23_tmp] += AlphaY_0[Tz23_tmp_tmp] * (real32_T)Tz23[i];
      Tz23_0[Tz23_tmp] += AlphaY_0[Tz23_tmp_tmp + 1] * (real32_T)Tz23[i + 4];
      Tz23_0[Tz23_tmp] += AlphaY_0[Tz23_tmp_tmp + 2] * (real32_T)Tz23[i + 8];
      Tz23_0[Tz23_tmp] += AlphaY_0[Tz23_tmp_tmp + 3] * (real32_T)Tz23[i + 12];
    }

    Tz23_tmp_tmp = i << 2;
    HTransform_tmp_3[Tz23_tmp_tmp] = HTransform_tmp_2[i];
    HTransform_tmp_3[Tz23_tmp_tmp + 3] = HTransform_tmp_1[i];
  }

  Green0_tmp_tmp[0] = 85;
  Green0_tmp_tmp[1] = 0;
  Green0_tmp_tmp[2] = 0;
  Green0_tmp_tmp[3] = 1;
  Yellow0_tmp[0] = -42.5;
  Yellow0_tmp[1] = 73.612159321677282;
  Yellow0_tmp[2] = 0.0;
  Yellow0_tmp[3] = 1.0;
  Blue0_tmp[0] = -42.5;
  Blue0_tmp[1] = -73.612159321677282;
  Blue0_tmp[2] = 0.0;
  Blue0_tmp[3] = 1.0;
  for (i = 0; i < 4; i++) {
    for (i_0 = 0; i_0 < 4; i_0++) {
      Tz23_tmp_tmp = i_0 << 2;
      Tz23_tmp = i + Tz23_tmp_tmp;
      AlphaY_0[Tz23_tmp] = 0.0F;
      AlphaY_0[Tz23_tmp] += HTransform_tmp_3[Tz23_tmp_tmp] * Tz23_0[i];
      AlphaY_0[Tz23_tmp] += HTransform_tmp_3[Tz23_tmp_tmp + 1] * Tz23_0[i + 4];
      AlphaY_0[Tz23_tmp] += HTransform_tmp_3[Tz23_tmp_tmp + 2] * Tz23_0[i + 8];
      AlphaY_0[Tz23_tmp] += HTransform_tmp_3[Tz23_tmp_tmp + 3] * Tz23_0[i + 12];
    }

    AlphaX = 0.0F;
    AlphaY = 0.0F;
    HTransform_tmp = 0.0F;
    for (i_0 = 0; i_0 < 4; i_0++) {
      Tz23_tmp_tmp = i_0 << 2;
      Tz23_tmp = i + Tz23_tmp_tmp;
      HTransform[Tz23_tmp] = 0.0F;
      HTransform[Tz23_tmp] += (real32_T)Tz23[Tz23_tmp_tmp] * AlphaY_0[i];
      HTransform[Tz23_tmp] += (real32_T)Tz23[Tz23_tmp_tmp + 1] * AlphaY_0[i + 4];
      HTransform[Tz23_tmp] += (real32_T)Tz23[Tz23_tmp_tmp + 2] * AlphaY_0[i + 8];
      HTransform[Tz23_tmp] += (real32_T)Tz23[Tz23_tmp_tmp + 3] * AlphaY_0[i + 12];
      AlphaX += HTransform[Tz23_tmp] * (real32_T)Green0_tmp_tmp[i_0];
      AlphaY += HTransform[Tz23_tmp] * (real32_T)Yellow0_tmp[i_0];
      HTransform_tmp += HTransform[Tz23_tmp] * (real32_T)Blue0_tmp[i_0];
    }

    Green0_tmp_tmp_0[i] = (real32_T)Green0_tmp_tmp[i] - AlphaX;
    Yellow0_tmp_0[i] = (real32_T)Yellow0_tmp[i] - AlphaY;
    Blue0_tmp_0[i] = (real32_T)Blue0_tmp[i] - HTransform_tmp;
  }

  AlphaX = regulator_nelin_P_B->Input3 * 3.14159274F / 180.0F;
  AlphaY = -regulator_nelin_P_B->Input4 * 3.14159274F / 180.0F;
  HTransform_tmp = sinf(AlphaY);
  AlphaY = cosf(AlphaY);
  HTransform_tmp_0 = sinf(AlphaX);
  AlphaX = cosf(AlphaX);
  AlphaY_0[0] = AlphaY;
  AlphaY_0[4] = 0.0F;
  AlphaY_0[8] = HTransform_tmp;
  AlphaY_0[12] = 0.0F;
  AlphaY_0[2] = -HTransform_tmp;
  AlphaY_0[6] = 0.0F;
  AlphaY_0[10] = AlphaY;
  AlphaY_0[14] = 0.0F;
  AlphaY_0[1] = 0.0F;
  AlphaY_0[3] = 0.0F;
  AlphaY_0[5] = 1.0F;
  AlphaY_0[7] = 0.0F;
  AlphaY_0[9] = 0.0F;
  AlphaY_0[11] = 0.0F;
  AlphaY_0[13] = 0.0F;
  AlphaY_0[15] = 1.0F;
  HTransform_tmp_3[1] = 0.0F;
  HTransform_tmp_3[5] = AlphaX;
  HTransform_tmp_3[9] = -HTransform_tmp_0;
  HTransform_tmp_3[13] = 0.0F;
  HTransform_tmp_3[2] = 0.0F;
  HTransform_tmp_3[6] = HTransform_tmp_0;
  HTransform_tmp_3[10] = AlphaX;
  HTransform_tmp_3[14] = 0.0F;
  for (i = 0; i < 4; i++) {
    for (i_0 = 0; i_0 < 4; i_0++) {
      Tz23_tmp_tmp = i_0 << 2;
      Tz23_tmp = i + Tz23_tmp_tmp;
      Tz23_0[Tz23_tmp] = 0.0F;
      Tz23_0[Tz23_tmp] += AlphaY_0[Tz23_tmp_tmp] * (real32_T)Tz23[i];
      Tz23_0[Tz23_tmp] += AlphaY_0[Tz23_tmp_tmp + 1] * (real32_T)Tz23[i + 4];
      Tz23_0[Tz23_tmp] += AlphaY_0[Tz23_tmp_tmp + 2] * (real32_T)Tz23[i + 8];
      Tz23_0[Tz23_tmp] += AlphaY_0[Tz23_tmp_tmp + 3] * (real32_T)Tz23[i + 12];
    }

    Tz23_tmp_tmp = i << 2;
    HTransform_tmp_3[Tz23_tmp_tmp] = HTransform_tmp_2[i];
    HTransform_tmp_3[Tz23_tmp_tmp + 3] = HTransform_tmp_1[i];
  }

  Yellow0_tmp[0] = -42.5;
  Yellow0_tmp[1] = 73.612159321677282;
  Yellow0_tmp[2] = 0.0;
  Yellow0_tmp[3] = 1.0;
  Blue0_tmp[0] = -42.5;
  Blue0_tmp[1] = -73.612159321677282;
  Blue0_tmp[2] = 0.0;
  Blue0_tmp[3] = 1.0;
  for (i = 0; i < 4; i++) {
    for (i_0 = 0; i_0 < 4; i_0++) {
      Tz23_tmp_tmp = i_0 << 2;
      Tz23_tmp = i + Tz23_tmp_tmp;
      AlphaY_0[Tz23_tmp] = 0.0F;
      AlphaY_0[Tz23_tmp] += HTransform_tmp_3[Tz23_tmp_tmp] * Tz23_0[i];
      AlphaY_0[Tz23_tmp] += HTransform_tmp_3[Tz23_tmp_tmp + 1] * Tz23_0[i + 4];
      AlphaY_0[Tz23_tmp] += HTransform_tmp_3[Tz23_tmp_tmp + 2] * Tz23_0[i + 8];
      AlphaY_0[Tz23_tmp] += HTransform_tmp_3[Tz23_tmp_tmp + 3] * Tz23_0[i + 12];
    }

    AlphaX = 0.0F;
    for (i_0 = 0; i_0 < 4; i_0++) {
      Tz23_tmp_tmp = i_0 << 2;
      Tz23_tmp = i + Tz23_tmp_tmp;
      HTransform[Tz23_tmp] = 0.0F;
      HTransform[Tz23_tmp] += (real32_T)Tz23[Tz23_tmp_tmp] * AlphaY_0[i];
      HTransform[Tz23_tmp] += (real32_T)Tz23[Tz23_tmp_tmp + 1] * AlphaY_0[i + 4];
      HTransform[Tz23_tmp] += (real32_T)Tz23[Tz23_tmp_tmp + 2] * AlphaY_0[i + 8];
      HTransform[Tz23_tmp] += (real32_T)Tz23[Tz23_tmp_tmp + 3] * AlphaY_0[i + 12];
      AlphaX += HTransform[Tz23_tmp] * (real32_T)Yellow0_tmp[i_0];
    }

    Yellow0_tmp_1[i] = (real32_T)Yellow0_tmp[i] - AlphaX;
  }

  /* Gain: '<Root>/Gain7' incorporates:
   *  Constant: '<S3>/cylinder height'
   *  Constant: '<S5>/cylinder height'
   *  Gain: '<Root>/Gain3'
   *  Gain: '<Root>/Gain5'
   *  Gain: '<S1>/Gain'
   *  Gain: '<S1>/Gain3'
   *  MATLAB Function: '<Root>/MATLAB Function'
   *  MATLAB Function: '<S1>/requested alfa 2 deltaz1'
   *  Sum: '<S3>/Sum'
   *  Sum: '<S5>/Sum'
   */
  regulator_nelin_P_B->Gain7 = (real32_T)(pow(2.71828182845904, (0.001F *
    regulator_nelin_P_norm(Yellow0_tmp_0, inst) - 0.115) * 1000.0 * 0.1528) * 0.03078
    - pow(2.71828182845904, (0.001F * regulator_nelin_P_norm(Yellow0_tmp_1, inst) -
    0.115) * 1000.0 * 0.1528) * 0.03078);

  /* S-Function (bur_out): '<Root>/Output1' */
  inst->Blue_tab = regulator_nelin_P_B->Gain7;

  /* MATLAB Function: '<S1>/requested alfa 2 deltaz1' */
  for (i = 0; i < 4; i++) {
    Yellow0_tmp_0[i] = (real32_T)Blue0_tmp[i] - ((HTransform[i + 4] *
      -73.6121597F + HTransform[i] * -42.5F) + HTransform[i + 12]);
  }

  /* Gain: '<Root>/Gain9' incorporates:
   *  Constant: '<S6>/cylinder height'
   *  Constant: '<S8>/cylinder height'
   *  Gain: '<Root>/Gain2'
   *  Gain: '<Root>/Gain6'
   *  Gain: '<S1>/Gain2'
   *  Gain: '<S1>/Gain5'
   *  MATLAB Function: '<Root>/MATLAB Function'
   *  MATLAB Function: '<S1>/requested alfa 2 deltaz1'
   *  Sum: '<S6>/Sum'
   *  Sum: '<S8>/Sum'
   */
  regulator_nelin_P_B->Gain9 = (real32_T)(pow(2.71828182845904, (0.001F *
    regulator_nelin_P_norm(Blue0_tmp_0, inst) - 0.115) * 1000.0 * 0.1528) * 0.03078 -
    pow(2.71828182845904, (0.001F * regulator_nelin_P_norm(Yellow0_tmp_0, inst) -
    0.115) * 1000.0 * 0.1528) * 0.03078);

  /* S-Function (bur_out): '<Root>/Output2' */
  inst->Yellow_tab = regulator_nelin_P_B->Gain9;

  /* MATLAB Function: '<S1>/requested alfa 2 deltaz1' */
  for (i = 0; i < 4; i++) {
    Blue0_tmp_0[i] = (real32_T)Green0_tmp_tmp[i] - (HTransform[i] * 85.0F +
      HTransform[i + 12]);
  }

  /* Gain: '<Root>/Gain8' incorporates:
   *  Constant: '<S4>/cylinder height'
   *  Constant: '<S7>/cylinder height'
   *  Gain: '<Root>/Gain1'
   *  Gain: '<Root>/Gain4'
   *  Gain: '<S1>/Gain1'
   *  Gain: '<S1>/Gain4'
   *  MATLAB Function: '<Root>/MATLAB Function'
   *  MATLAB Function: '<S1>/requested alfa 2 deltaz1'
   *  Sum: '<S4>/Sum'
   *  Sum: '<S7>/Sum'
   */
  regulator_nelin_P_B->Gain8 = (real32_T)(pow(2.71828182845904, (0.001F *
    regulator_nelin_P_norm(Green0_tmp_tmp_0, inst) - 0.115) * 1000.0 * 0.1528) *
    0.03078 - pow(2.71828182845904, (0.001F * regulator_nelin_P_norm(Blue0_tmp_0, inst)
    - 0.115) * 1000.0 * 0.1528) * 0.03078);

  /* S-Function (bur_out): '<Root>/Output4' */
  inst->Green_tab = regulator_nelin_P_B->Gain8;
}

/* Model initialize function */
void regulator_nelin_P_initialize(RT_MODEL_regulator_nelin_P_T *const
  regulator_nelin_P_M, struct nonL_P* inst)
{
  UNUSED_PARAMETER(regulator_nelin_P_M);
}

/* Model terminate function */
void regulator_nelin_P_terminate(RT_MODEL_regulator_nelin_P_T
  * regulator_nelin_P_M, struct nonL_P* inst)
{}

/* Model data allocation function */
void regulator_nelin_P_initializeMemory(RT_MODEL_regulator_nelin_P_T* const regulator_nelin_P_M, struct nonL_P * inst)
{
  /* block I/O */
  {
  }

  {
    B_regulator_nelin_P_T *regulator_nelin_P_B = regulator_nelin_P_M->blockIO;

    /* block I/O */
    {
      regulator_nelin_P_B->Input1 = 0.0F;
      regulator_nelin_P_B->Input2 = 0.0F;
      regulator_nelin_P_B->Input3 = 0.0F;
      regulator_nelin_P_B->Input4 = 0.0F;
      regulator_nelin_P_B->Gain7 = 0.0F;
      regulator_nelin_P_B->Gain9 = 0.0F;
      regulator_nelin_P_B->Gain8 = 0.0F;
    }
  }

}
```

### Program Logical/Source/Program (IEC)

#### Variables.var
```iecst
VAR
	TON_0 : TON;
	TON_1 : TON;
	TON_2 : TON;
	TON_3 : TON;
	TON_4 : TON;
	i : INT;
END_VAR
```

#### Cyclic.st
```iecst
PROGRAM _CYCLIC

	TON_0(IN := automatika.casovac, PT := INT_TO_TIME(automatika.cas));
	TON_1(IN := automatika.casovac_uchopenie, PT := T#4s);
	//TON_2(IN := automatika.trajectoryStart, PT := automatika.trajectoryTime);
	//TON_4(IN := automatika.trajectoryStart2, PT := automatika.trajectoryTime2);
	//TON_3(IN := automatika.novyCyklusStart, PT := automatika.novyCyklus);

	CASE global_step OF

		0:	// caka kym spravi uvodne odmeranie referencii....v controlleri ak je krok 4, vtedy prechadza global_step = 1
			(*
			automatika.y_desired[0]	:= 0;
			automatika.y_desired[1]	:= 0;
			automatika.y_desired[2]	:= 0;
			automatika.y_desired[3]	:= 0;
			automatika.y_desired[4]	:= 0;
			automatika.y_desired[5]	:= 0;
			automatika.y_desired[6]	:= 0;

			automatika.x_desired[0]	:= 0;
			automatika.x_desired[1]	:= 0;
			automatika.x_desired[2]	:= 0;
			automatika.x_desired[3]	:= 0;
			automatika.x_desired[4]	:= 0;
			automatika.x_desired[5]	:= 0;
			automatika.x_desired[6]	:= 0;
			*)
			automatika.linear		:= 23;
			FOR i:=0 TO 6 BY 1 DO
				automatika.I_konstanta[i]	:= 5;
			END_FOR
			automatika.automatic	:= FALSE;
			(*
			IF automatika.step_color = 1 OR automatika.step_color = 2 THEN
				global_step				:= 999;
			END_IF
			*)
			modul;

		999:
			IF automatika.step_color = 1 OR automatika.step_color = 2 THEN
				automatika.loptickyVzasobniku	:= TRUE;
			ELSE
				automatika.loptickyVzasobniku	:= FALSE;
			END_IF

			IF automatika.loptickyVzasobniku = TRUE OR global_step_udp = 1 THEN
				automatika.effector		:= FALSE;
			//	global_step_udp			:= 0;
				global_step				:= 1;
				automatika.automatic	:= FALSE;
				I_ON					:= FALSE;
			END_IF
			FOR i:=0 TO 6 BY 1 DO
				automatika.I_konstanta[i]	:= 0;
			END_FOR

		1:
			automatika.cas			:= 1000;
			automatika.casovac		:= TRUE;
			I_ON					:= TRUE;
			global_step				:= 100;

		100:
			IF TON_0.Q = TRUE THEN
				automatika.casovac	:= FALSE;
				IF global_step_udp = 1 THEN
					global_step				:= 11;
				ELSE
					automatika.cas			:= 1000;
					automatika.casovac		:= TRUE;
					global_step				:= 2;
				END_IF
			END_IF

		2:
			IF TON_0.Q=TRUE THEN
				automatika.casovac		:= FALSE;
				//automatika.ball_up		:= TRUE;
				global_step				:= 3;
			//	automatika.ball_piston	:= FALSE;
			END_IF

		3:	// pohyb pre uchopenie gulicky
			//automatika.casovac_uchopenie	:= TRUE;
			IF(automatika.step_color = 1)THEN
				automatika.box := 1;
				automatika.loptickyVzasobniku := TRUE;
			ELSIF(automatika.step_color = 2)THEN
				automatika.box	:= 2;
				automatika.loptickyVzasobniku := TRUE;
			ELSIF(automatika.step_color = 3)THEN
				automatika.loptickyVzasobniku := FALSE;
				automatika.box := 3;
			END_IF

			automatika.casovac			:= TRUE;
			automatika.cas				:= 5000;
			automatika.effector			:= FALSE;
			automatika.linear			:= 23;
			global_step					:= 4;
			FOR i:=0 TO 6 BY 1 DO
				automatika.I_konstanta[i]	:= 30;
			END_FOR
		4:
			// Pohyb ku levitujucej lopte

			automatika.y_desired[0]	:= TIME_TO_INT(TON_0.ET)*(-7)/((automatika.cas));
			automatika.y_desired[1]	:= TIME_TO_INT(TON_0.ET)*(6)/((automatika.cas));
			automatika.y_desired[2]	:= TIME_TO_INT(TON_0.ET)*(-10)/((automatika.cas));
			automatika.y_desired[3]	:= TIME_TO_INT(TON_0.ET)*(-10)/((automatika.cas));
			automatika.y_desired[4]	:= TIME_TO_INT(TON_0.ET)*(-8)/((automatika.cas));
			automatika.y_desired[5]	:= TIME_TO_INT(TON_0.ET)*(-5)/((automatika.cas));
			automatika.y_desired[6]	:= TIME_TO_INT(TON_0.ET)*(-5)/((automatika.cas));//-10

			automatika.x_desired[0]	:= TIME_TO_INT(TON_0.ET)*5/((automatika.cas));
			automatika.x_desired[1]	:= TIME_TO_INT(TON_0.ET)*4/((automatika.cas));
			automatika.x_desired[2]	:= TIME_TO_INT(TON_0.ET)*5/((automatika.cas));
			automatika.x_desired[3]	:= TIME_TO_INT(TON_0.ET)*5/((automatika.cas));
			automatika.x_desired[4]	:= TIME_TO_INT(TON_0.ET)*5/((automatika.cas));
			automatika.x_desired[5]	:= TIME_TO_INT(TON_0.ET)*1/((automatika.cas));
			automatika.x_desired[6]	:= 0;// TIME_TO_INT(TON_0.ET)*2/((automatika.cas));

			//automatika.linear		:= TIME_TO_INT(TON_2.ET)*30/(TIME_TO_INT(automatika.trajectoryTime));

			IF TON_0.Q=TRUE THEN
				automatika.casovac			:= FALSE;
				automatika.casovac_uchopenie:= TRUE;
				global_step					:= 55;
				FOR i:=0 TO 6 BY 1 DO
					automatika.x_desired_previous[i]	:= automatika.x_desired[i];
					automatika.y_desired_previous[i]	:= automatika.y_desired[i];
					automatika.I_konstanta[i]			:= 20;
				END_FOR
			END_IF

		55:
			IF TON_1.Q = TRUE THEN
				automatika.levitacia			:= TRUE;
				automatika.linear				:= 30;
				automatika.casovac_uchopenie	:= FALSE;
				global_step						:= 555;
			END_IF

		555:
			automatika.cas						:= 1000;
			automatika.casovac					:= TRUE;
			global_step							:= 5;

		5:	// uchopenie
			IF TON_0.Q = TRUE THEN
				automatika.casovac				:= FALSE;
				automatika.effector				:= TRUE;
				global_step						:= 6;
			END_IF

		6:
			automatika.casovac_uchopenie		:= TRUE;
			global_step							:= 7;
			automatika.linear					:= 23;

		7:
			IF TON_1.Q = TRUE THEN
				automatika.casovac_uchopenie	:= FALSE;
				global_step						:= 8;
				automatika.levitacia			:= FALSE;
				automatika.ball_piston			:= TRUE;
				automatika.cas					:= 4500;
				automatika.casovac				:= TRUE;
				FOR i:=0 TO 6 BY 1 DO
					automatika.I_konstanta[i]	:= 50;
				END_FOR
			END_IF

		8:
			IF(automatika.box = 1) THEN
				// prenesenie objektu
				automatika.y_desired[0]	:= (automatika.y_desired_previous[0]*(automatika.cas - TIME_TO_INT(TON_0.ET))/automatika.cas) + TIME_TO_INT(TON_0.ET)*(7)/((automatika.cas));
				automatika.y_desired[1]	:= (automatika.y_desired_previous[1]*(automatika.cas - TIME_TO_INT(TON_0.ET))/automatika.cas) +  TIME_TO_INT(TON_0.ET)*(0)/((automatika.cas));	// 5000ms
				automatika.y_desired[2]	:= (automatika.y_desired_previous[2]*(automatika.cas - TIME_TO_INT(TON_0.ET))/automatika.cas) +  TIME_TO_INT(TON_0.ET)*(10)/((automatika.cas));
				automatika.y_desired[3]	:= (automatika.y_desired_previous[3]*(automatika.cas - TIME_TO_INT(TON_0.ET))/automatika.cas) +  TIME_TO_INT(TON_0.ET)*(0)/((automatika.cas));
				automatika.y_desired[4]	:= (automatika.y_desired_previous[4]*(automatika.cas - TIME_TO_INT(TON_0.ET))/automatika.cas) +  TIME_TO_INT(TON_0.ET)*(8)/((automatika.cas));
				automatika.y_desired[5]	:= (automatika.y_desired_previous[5]*(automatika.cas - TIME_TO_INT(TON_0.ET))/automatika.cas) +  TIME_TO_INT(TON_0.ET)*(5)/((automatika.cas));
				automatika.y_desired[6]	:= (automatika.y_desired_previous[6]*(automatika.cas - TIME_TO_INT(TON_0.ET))/automatika.cas) +  TIME_TO_INT(TON_0.ET)*(10)/((automatika.cas));

				automatika.x_desired[0]	:= (automatika.x_desired_previous[0]*(automatika.cas - TIME_TO_INT(TON_0.ET))/automatika.cas) +  TIME_TO_INT(TON_0.ET)*(2)/((automatika.cas));
				automatika.x_desired[1]	:= (automatika.x_desired_previous[1]*(automatika.cas - TIME_TO_INT(TON_0.ET))/automatika.cas) +  TIME_TO_INT(TON_0.ET)*(-2)/((automatika.cas));
				automatika.x_desired[2]	:= (automatika.x_desired_previous[2]*(automatika.cas - TIME_TO_INT(TON_0.ET))/automatika.cas) +  TIME_TO_INT(TON_0.ET)*(-2)/((automatika.cas));
				automatika.x_desired[3]	:= (automatika.x_desired_previous[3]*(automatika.cas - TIME_TO_INT(TON_0.ET))/automatika.cas) +  TIME_TO_INT(TON_0.ET)*(-2)/((automatika.cas));
				automatika.x_desired[4]	:= (automatika.x_desired_previous[4]*(automatika.cas - TIME_TO_INT(TON_0.ET))/automatika.cas) +  TIME_TO_INT(TON_0.ET)*(-5)/((automatika.cas));
				automatika.x_desired[5]	:= (automatika.x_desired_previous[5]*(automatika.cas - TIME_TO_INT(TON_0.ET))/automatika.cas) +  TIME_TO_INT(TON_0.ET)*(-5)/((automatika.cas));
				automatika.x_desired[6]	:= TIME_TO_INT(TON_0.ET)*(-5)/((automatika.cas));

				automatika.linear		:= TIME_TO_INT(TON_0.ET)*30/((automatika.cas));
			ELSIF(automatika.box = 2) THEN
				// prenesenie objektu
				automatika.y_desired[0]	:= (automatika.y_desired_previous[0]*(automatika.cas - TIME_TO_INT(TON_0.ET))/automatika.cas) + TIME_TO_INT(TON_0.ET)*(7)/((automatika.cas));
				automatika.y_desired[1]	:= (automatika.y_desired_previous[1]*(automatika.cas - TIME_TO_INT(TON_0.ET))/automatika.cas) + TIME_TO_INT(TON_0.ET)*(2)/((automatika.cas));	// 5000ms
				automatika.y_desired[2]	:= (automatika.y_desired_previous[2]*(automatika.cas - TIME_TO_INT(TON_0.ET))/automatika.cas) + TIME_TO_INT(TON_0.ET)*(10)/((automatika.cas));
				automatika.y_desired[3]	:= (automatika.y_desired_previous[3]*(automatika.cas - TIME_TO_INT(TON_0.ET))/automatika.cas) + TIME_TO_INT(TON_0.ET)*(0)/((automatika.cas));
				automatika.y_desired[4]	:= (automatika.y_desired_previous[4]*(automatika.cas - TIME_TO_INT(TON_0.ET))/automatika.cas) + TIME_TO_INT(TON_0.ET)*(8)/((automatika.cas));
				automatika.y_desired[5]	:= (automatika.y_desired_previous[5]*(automatika.cas - TIME_TO_INT(TON_0.ET))/automatika.cas) + TIME_TO_INT(TON_0.ET)*(5)/((automatika.cas));
				automatika.y_desired[6]	:= (automatika.y_desired_previous[6]*(automatika.cas - TIME_TO_INT(TON_0.ET))/automatika.cas) + TIME_TO_INT(TON_0.ET)*(10)/((automatika.cas));

				automatika.x_desired[0]	:= (automatika.x_desired_previous[0]*(automatika.cas - TIME_TO_INT(TON_0.ET))/automatika.cas) + TIME_TO_INT(TON_0.ET)*(-8)/((automatika.cas));//-5
				automatika.x_desired[1]	:= (automatika.x_desired_previous[1]*(automatika.cas - TIME_TO_INT(TON_0.ET))/automatika.cas) + TIME_TO_INT(TON_0.ET)*(-3)/((automatika.cas));//0
				automatika.x_desired[2]	:= (automatika.x_desired_previous[2]*(automatika.cas - TIME_TO_INT(TON_0.ET))/automatika.cas) + TIME_TO_INT(TON_0.ET)*(5)/((automatika.cas));
				automatika.x_desired[3]	:= (automatika.x_desired_previous[3]*(automatika.cas - TIME_TO_INT(TON_0.ET))/automatika.cas) + TIME_TO_INT(TON_0.ET)*(10)/((automatika.cas));
				automatika.x_desired[4]	:= (automatika.x_desired_previous[4]*(automatika.cas - TIME_TO_INT(TON_0.ET))/automatika.cas) + TIME_TO_INT(TON_0.ET)*(10)/((automatika.cas));
				automatika.x_desired[5]	:= (automatika.x_desired_previous[5]*(automatika.cas - TIME_TO_INT(TON_0.ET))/automatika.cas) + TIME_TO_INT(TON_0.ET)*(0)/((automatika.cas));
				automatika.x_desired[6]	:= 0;

				automatika.linear		:= TIME_TO_INT(TON_0.ET)*30/((automatika.cas));
			ELSIF(automatika.box = 3) THEN
				(*
				IF(automatika.step_color = 1)THEN
					automatika.loptickyVzasobniku	:= TRUE;
					automatika.box := 1;
				ELSIF(automatika.step_color = 2)THEN
					automatika.box	:= 2;
					automatika.loptickyVzasobniku	:= TRUE;
				ELSIF(automatika.step_color = 3)THEN
					*)
					automatika.y_desired[0]	:= (automatika.y_desired_previous[0]*(automatika.cas - TIME_TO_INT(TON_0.ET))/automatika.cas);//+ TIME_TO_INT(TON_0.ET)*(1)/((automatika.cas));
					automatika.y_desired[1]	:= (automatika.y_desired_previous[1]*(automatika.cas - TIME_TO_INT(TON_0.ET))/automatika.cas);//TIME_TO_INT(TON_0.ET)*(1)/((automatika.cas));	// 5000ms
					automatika.y_desired[2]	:= (automatika.y_desired_previous[2]*(automatika.cas - TIME_TO_INT(TON_0.ET))/automatika.cas);// TIME_TO_INT(TON_0.ET)*(1)/((automatika.cas));
					automatika.y_desired[3]	:= (automatika.y_desired_previous[3]*(automatika.cas - TIME_TO_INT(TON_0.ET))/automatika.cas);//TIME_TO_INT(TON_0.ET)*(1)/((automatika.cas));
					automatika.y_desired[4]	:= (automatika.y_desired_previous[4]*(automatika.cas - TIME_TO_INT(TON_0.ET))/automatika.cas);//TIME_TO_INT(TON_0.ET)*(1)/((automatika.cas));
					automatika.y_desired[5]	:= (automatika.y_desired_previous[5]*(automatika.cas - TIME_TO_INT(TON_0.ET))/automatika.cas);//TIME_TO_INT(TON_0.ET)*(1)/((automatika.cas));
					automatika.y_desired[6]	:= (automatika.y_desired_previous[6]*(automatika.cas - TIME_TO_INT(TON_0.ET))/automatika.cas);//TIME_TO_INT(TON_0.ET)*(1)/((automatika.cas));

					automatika.x_desired[0]	:= (automatika.x_desired_previous[0]*(automatika.cas - TIME_TO_INT(TON_0.ET))/automatika.cas);//TIME_TO_INT(TON_0.ET)*(1)/((automatika.cas));
					automatika.x_desired[1]	:= (automatika.x_desired_previous[1]*(automatika.cas - TIME_TO_INT(TON_0.ET))/automatika.cas);//TIME_TO_INT(TON_0.ET)*(1)/((automatika.cas));
					automatika.x_desired[2]	:= (automatika.x_desired_previous[2]*(automatika.cas - TIME_TO_INT(TON_0.ET))/automatika.cas);//TIME_TO_INT(TON_0.ET)*(1)/((automatika.cas));
					automatika.x_desired[3]	:= (automatika.x_desired_previous[3]*(automatika.cas - TIME_TO_INT(TON_0.ET))/automatika.cas);//TIME_TO_INT(TON_0.ET)*(1)/((automatika.cas));
					automatika.x_desired[4]	:= (automatika.x_desired_previous[4]*(automatika.cas - TIME_TO_INT(TON_0.ET))/automatika.cas);//TIME_TO_INT(TON_0.ET)*(1)/((automatika.cas));
					automatika.x_desired[5]	:= (automatika.x_desired_previous[5]*(automatika.cas - TIME_TO_INT(TON_0.ET))/automatika.cas);//TIME_TO_INT(TON_0.ET)*(1)/((automatika.cas));
					automatika.x_desired[6]	:= 0;//TIME_TO_INT(TON_0.ET)*(1)/((automatika.cas));;

					automatika.loptickyVzasobniku	:= FALSE;
					automatika.effector				:= FALSE;
					global_step						:= 0;
				//END_IF

			END_IF

			IF TON_0.Q=TRUE THEN
				automatika.casovac					:= FALSE;
				automatika.ball_piston				:= FALSE;
				automatika.loptickyVzasobniku		:= TRUE;		// pridane 15.11.2024
				IF automatika.loptickyVzasobniku = TRUE THEN
					global_step						:= 9;
				ELSE
					global_step						:= 999;//0
				END_IF
				FOR i:=0 TO 6 BY 1 DO
					automatika.x_desired_previous[i]:= automatika.x_desired[i];
					automatika.y_desired_previous[i]:= automatika.y_desired[i];
				END_FOR
			END_IF

		9:
			automatika.effector				:= FALSE;
			automatika.cas					:= 2000;
			automatika.casovac				:= TRUE;
			global_step						:= 901;

		901:
			IF(automatika.step_color = 3)THEN
				automatika.testFarba	:= 1;
			END_IF
			global_step					:= 902;

		902:
			IF(automatika.step_color = 3)THEN
				automatika.testFarba	:= 2;
			END_IF
			global_step					:= 903;

		903:
			IF TON_0.Q = TRUE THEN
				automatika.casovac			:= FALSE;
				automatika.popcorn			:= FALSE;
				IF(automatika.step_color = 3)THEN
					automatika.testFarba	:= 0;
					automatika.loptickyVzasobniku	:= FALSE;
				END_IF
				global_step					:= 904;
			END_IF

		904:
			automatika.cas					:= 4000;
			automatika.casovac				:= TRUE;
			global_step						:= 905;

		905:

			automatika.y_desired[0]	:= (automatika.y_desired_previous[0]*(automatika.cas - TIME_TO_INT(TON_0.ET))/automatika.cas) + TIME_TO_INT(TON_0.ET)*(1)/((automatika.cas));
			automatika.y_desired[1]	:= (automatika.y_desired_previous[1]*(automatika.cas - TIME_TO_INT(TON_0.ET))/automatika.cas) + TIME_TO_INT(TON_0.ET)*(1)/((automatika.cas));	// 5000ms
			automatika.y_desired[2]	:= (automatika.y_desired_previous[2]*(automatika.cas - TIME_TO_INT(TON_0.ET))/automatika.cas) + TIME_TO_INT(TON_0.ET)*(1)/((automatika.cas));
			automatika.y_desired[3]	:= (automatika.y_desired_previous[3]*(automatika.cas - TIME_TO_INT(TON_0.ET))/automatika.cas) + TIME_TO_INT(TON_0.ET)*(1)/((automatika.cas));
			automatika.y_desired[4]	:= (automatika.y_desired_previous[4]*(automatika.cas - TIME_TO_INT(TON_0.ET))/automatika.cas) + TIME_TO_INT(TON_0.ET)*(1)/((automatika.cas));
			automatika.y_desired[5]	:= (automatika.y_desired_previous[5]*(automatika.cas - TIME_TO_INT(TON_0.ET))/automatika.cas) + TIME_TO_INT(TON_0.ET)*(1)/((automatika.cas));
			automatika.y_desired[6]	:= (automatika.y_desired_previous[6]*(automatika.cas - TIME_TO_INT(TON_0.ET))/automatika.cas) + TIME_TO_INT(TON_0.ET)*(1)/((automatika.cas));

			automatika.x_desired[0]	:= (automatika.x_desired_previous[0]*(automatika.cas - TIME_TO_INT(TON_0.ET))/automatika.cas) + TIME_TO_INT(TON_0.ET)*(1)/((automatika.cas));
			automatika.x_desired[1]	:= (automatika.x_desired_previous[1]*(automatika.cas - TIME_TO_INT(TON_0.ET))/automatika.cas) + TIME_TO_INT(TON_0.ET)*(1)/((automatika.cas));
			automatika.x_desired[2]	:= (automatika.x_desired_previous[2]*(automatika.cas - TIME_TO_INT(TON_0.ET))/automatika.cas) + TIME_TO_INT(TON_0.ET)*(1)/((automatika.cas));
			automatika.x_desired[3]	:= (automatika.x_desired_previous[3]*(automatika.cas - TIME_TO_INT(TON_0.ET))/automatika.cas) + TIME_TO_INT(TON_0.ET)*(1)/((automatika.cas));
			automatika.x_desired[4]	:= (automatika.x_desired_previous[4]*(automatika.cas - TIME_TO_INT(TON_0.ET))/automatika.cas) + TIME_TO_INT(TON_0.ET)*(1)/((automatika.cas));
			automatika.x_desired[5]	:= (automatika.x_desired_previous[5]*(automatika.cas - TIME_TO_INT(TON_0.ET))/automatika.cas) + TIME_TO_INT(TON_0.ET)*(1)/((automatika.cas));
			automatika.x_desired[6]	:= (automatika.x_desired_previous[6]*(automatika.cas - TIME_TO_INT(TON_0.ET))/automatika.cas) + TIME_TO_INT(TON_0.ET)*(1)/((automatika.cas));

			automatika.linear		:= 23;

			IF TON_0.Q = TRUE THEN
				automatika.casovac			:= FALSE;
				global_step					:= 999;//posledne bolo 1 predtym 0
			END_IF

		11:
			automatika.cas					:= 5000;
			global_step						:= 111;
			automatika.linear				:= 23;
			FOR i:=0 TO 6 BY 1 DO
				automatika.x_desired_previous[i]:= automatika.x_desired[i];
				automatika.y_desired_previous[i]:= automatika.y_desired[i];
				automatika.I_konstanta[i]	:= 50;
			END_FOR
			automatika.casovac				:= TRUE;

		111:
			// ide po loptu
			automatika.y_desired[0]	:= (automatika.y_desired_previous[0]*(automatika.cas - TIME_TO_INT(TON_0.ET))/automatika.cas) + TIME_TO_INT(TON_0.ET)*(2)/((automatika.cas));//0
			automatika.y_desired[1]	:= (automatika.y_desired_previous[1]*(automatika.cas - TIME_TO_INT(TON_0.ET))/automatika.cas) + TIME_TO_INT(TON_0.ET)*(18)/((automatika.cas));
			automatika.y_desired[2]	:= (automatika.y_desired_previous[2]*(automatika.cas - TIME_TO_INT(TON_0.ET))/automatika.cas) + TIME_TO_INT(TON_0.ET)*(18)/((automatika.cas));
			automatika.y_desired[3]	:= (automatika.y_desired_previous[3]*(automatika.cas - TIME_TO_INT(TON_0.ET))/automatika.cas) + TIME_TO_INT(TON_0.ET)*(18)/((automatika.cas));
			automatika.y_desired[4]	:= (automatika.y_desired_previous[4]*(automatika.cas - TIME_TO_INT(TON_0.ET))/automatika.cas) + TIME_TO_INT(TON_0.ET)*(-18)/((automatika.cas));
			automatika.y_desired[5]	:= (automatika.y_desired_previous[5]*(automatika.cas - TIME_TO_INT(TON_0.ET))/automatika.cas) + TIME_TO_INT(TON_0.ET)*(-15)/((automatika.cas));
			automatika.y_desired[6]	:= (automatika.y_desired_previous[6]*(automatika.cas - TIME_TO_INT(TON_0.ET))/automatika.cas) + TIME_TO_INT(TON_0.ET)*(-18)/((automatika.cas));//-18

			automatika.x_desired[0]	:= (automatika.x_desired_previous[0]*(automatika.cas - TIME_TO_INT(TON_0.ET))/automatika.cas) + TIME_TO_INT(TON_0.ET)*(15)/((automatika.cas));
			automatika.x_desired[1]	:= (automatika.x_desired_previous[1]*(automatika.cas - TIME_TO_INT(TON_0.ET))/automatika.cas) + TIME_TO_INT(TON_0.ET)*(13)/((automatika.cas));
			automatika.x_desired[2]	:= (automatika.x_desired_previous[2]*(automatika.cas - TIME_TO_INT(TON_0.ET))/automatika.cas) + TIME_TO_INT(TON_0.ET)*(3)/((automatika.cas));
			automatika.x_desired[3]	:= (automatika.x_desired_previous[3]*(automatika.cas - TIME_TO_INT(TON_0.ET))/automatika.cas) + TIME_TO_INT(TON_0.ET)*(10)/((automatika.cas));
			automatika.x_desired[4]	:= (automatika.x_desired_previous[4]*(automatika.cas - TIME_TO_INT(TON_0.ET))/automatika.cas) + TIME_TO_INT(TON_0.ET)*(-10)/((automatika.cas));
			automatika.x_desired[5]	:= (automatika.x_desired_previous[5]*(automatika.cas - TIME_TO_INT(TON_0.ET))/automatika.cas) + TIME_TO_INT(TON_0.ET)*(-12)/((automatika.cas));
			automatika.x_desired[6]	:= (automatika.x_desired_previous[6]*(automatika.cas - TIME_TO_INT(TON_0.ET))/automatika.cas) + TIME_TO_INT(TON_0.ET)*(-15)/((automatika.cas));//-10

			IF TON_0.Q=TRUE THEN
				automatika.casovac			:= FALSE;
				global_step					:= 1110;
			END_IF
		1110:
			automatika.cas					:= 3500;
			automatika.casovac				:= TRUE;
			global_step						:= 11101;
		11101:
			IF TON_0.Q = TRUE THEN
				automatika.casovac			:= FALSE;
				automatika.ball_up			:= TRUE;
				global_step					:= 11102;
			END_IF
		11102:
			automatika.cas					:= 3000;
			automatika.casovac				:= TRUE;
			global_step						:= 1112;

		1112:// pockanie na vysunutie linearneho clena
			IF TON_0.Q = TRUE THEN
				automatika.casovac		:= FALSE;
			//	automatika.linear		:= 30;
				global_step				:= 1113;
			END_IF

		1113:// uchopenie lopty
			automatika.cas				:= 3000;
			automatika.casovac			:= TRUE;
			automatika.effector			:= TRUE;
			global_step					:= 122;

		122://pockanie na uchopenie lopty
			IF TON_0.Q = TRUE THEN
				automatika.casovac			:= FALSE;
				automatika.linear			:= 23;
				automatika.ball_up			:= FALSE;	// dvihac lopty dole
				global_step					:= 1222;
			END_IF

		1222:
			automatika.cas					:= 3000;
			automatika.casovac				:= TRUE;
			global_step						:= 12222;
		12222:
			IF TON_0.Q = TRUE THEN
				automatika.casovac			:= FALSE;
				global_step					:= 12223;
			END_IF

		12223:
			automatika.cas					:= 3000;
			automatika.casovac				:= TRUE;

			FOR i:=0 TO 6 BY 1 DO
				automatika.x_desired_previous[i]:= automatika.x_desired[i];
				automatika.y_desired_previous[i]:= automatika.y_desired[i];
			END_FOR
			global_step						:= 12224;

		12224:

			// nulova poloha
			automatika.y_desired[0]	:= (automatika.y_desired_previous[0]*(automatika.cas - TIME_TO_INT(TON_0.ET))/automatika.cas) + TIME_TO_INT(TON_0.ET)*(1)/((automatika.cas));
			automatika.y_desired[1]	:= (automatika.y_desired_previous[1]*(automatika.cas - TIME_TO_INT(TON_0.ET))/automatika.cas) + TIME_TO_INT(TON_0.ET)*(1)/((automatika.cas));
			automatika.y_desired[2]	:= (automatika.y_desired_previous[2]*(automatika.cas - TIME_TO_INT(TON_0.ET))/automatika.cas) + TIME_TO_INT(TON_0.ET)*(1)/((automatika.cas));
			automatika.y_desired[3]	:= (automatika.y_desired_previous[3]*(automatika.cas - TIME_TO_INT(TON_0.ET))/automatika.cas) + TIME_TO_INT(TON_0.ET)*(1)/((automatika.cas));
			(*
			automatika.y_desired[4]	:= TIME_TO_INT(TON_0.ET)*(0)/((automatika.cas));
			automatika.y_desired[5]	:= TIME_TO_INT(TON_0.ET)*(0)/((automatika.cas));
			automatika.y_desired[6]	:= TIME_TO_INT(TON_0.ET)*(0)/((automatika.cas));

			automatika.x_desired[0]	:= TIME_TO_INT(TON_0.ET)*(-12)/((automatika.cas));
			automatika.x_desired[1]	:= TIME_TO_INT(TON_0.ET)*(-10)/((automatika.cas));
			automatika.x_desired[2]	:= TIME_TO_INT(TON_0.ET)*(10)/((automatika.cas));
			automatika.x_desired[3]	:= TIME_TO_INT(TON_0.ET)*(10)/((automatika.cas));
			automatika.x_desired[4]	:= TIME_TO_INT(TON_0.ET)*(15)/((automatika.cas));
			automatika.x_desired[5]	:= TIME_TO_INT(TON_0.ET)*(15)/((automatika.cas));
			automatika.x_desired[6]	:= TIME_TO_INT(TON_0.ET)*(15)/((automatika.cas));
			*)
			IF TON_0.Q = TRUE THEN
				automatika.casovac			:= FALSE;
				global_step					:= 12225;
			END_IF

		12225:
			automatika.cas					:= 4000;
			FOR i:=0 TO 6 BY 1 DO
				automatika.x_desired_previous[i]:= automatika.x_desired[i];
				automatika.y_desired_previous[i]:= automatika.y_desired[i];
			END_FOR
			automatika.casovac				:= TRUE;
			automatika.popcorn				:= TRUE;
			global_step						:= 12226;

		12226:
			(*
			automatika.x_desired[0]	:= TIME_TO_INT(TON_0.ET)*(1)/((automatika.cas));
			automatika.x_desired[1]	:= TIME_TO_INT(TON_0.ET)*(1)/((automatika.cas));
			automatika.x_desired[2]	:= TIME_TO_INT(TON_0.ET)*(1)/((automatika.cas));
			automatika.x_desired[3]	:= TIME_TO_INT(TON_0.ET)*(1)/((automatika.cas));
			automatika.x_desired[4]	:= TIME_TO_INT(TON_0.ET)*(1)/((automatika.cas));
			automatika.x_desired[5]	:= TIME_TO_INT(TON_0.ET)*(1)/((automatika.cas));
			automatika.x_desired[6]	:= TIME_TO_INT(TON_0.ET)*(1)/((automatika.cas));
			*)

			automatika.y_desired[0]	:= (automatika.y_desired_previous[0]*(automatika.cas - TIME_TO_INT(TON_0.ET))/automatika.cas) + TIME_TO_INT(TON_0.ET)*(1)/((automatika.cas));
			automatika.y_desired[1]	:= (automatika.y_desired_previous[1]*(automatika.cas - TIME_TO_INT(TON_0.ET))/automatika.cas) + TIME_TO_INT(TON_0.ET)*(1)/((automatika.cas));	// 5000ms
			automatika.y_desired[2]	:= (automatika.y_desired_previous[2]*(automatika.cas - TIME_TO_INT(TON_0.ET))/automatika.cas) + TIME_TO_INT(TON_0.ET)*(1)/((automatika.cas));
			automatika.y_desired[3]	:= (automatika.y_desired_previous[3]*(automatika.cas - TIME_TO_INT(TON_0.ET))/automatika.cas) + TIME_TO_INT(TON_0.ET)*(1)/((automatika.cas));
			automatika.y_desired[4]	:= (automatika.y_desired_previous[4]*(automatika.cas - TIME_TO_INT(TON_0.ET))/automatika.cas) + TIME_TO_INT(TON_0.ET)*(1)/((automatika.cas));
			automatika.y_desired[5]	:= (automatika.y_desired_previous[5]*(automatika.cas - TIME_TO_INT(TON_0.ET))/automatika.cas) + TIME_TO_INT(TON_0.ET)*(1)/((automatika.cas));
			automatika.y_desired[6]	:= (automatika.y_desired_previous[6]*(automatika.cas - TIME_TO_INT(TON_0.ET))/automatika.cas) + TIME_TO_INT(TON_0.ET)*(1)/((automatika.cas));

			automatika.x_desired[0]	:= (automatika.x_desired_previous[0]*(automatika.cas - TIME_TO_INT(TON_0.ET))/automatika.cas) + TIME_TO_INT(TON_0.ET)*(1)/((automatika.cas));
			automatika.x_desired[1]	:= (automatika.x_desired_previous[1]*(automatika.cas - TIME_TO_INT(TON_0.ET))/automatika.cas) + TIME_TO_INT(TON_0.ET)*(1)/((automatika.cas));
			automatika.x_desired[2]	:= (automatika.x_desired_previous[2]*(automatika.cas - TIME_TO_INT(TON_0.ET))/automatika.cas) + TIME_TO_INT(TON_0.ET)*(1)/((automatika.cas));
			automatika.x_desired[3]	:= (automatika.x_desired_previous[3]*(automatika.cas - TIME_TO_INT(TON_0.ET))/automatika.cas) + TIME_TO_INT(TON_0.ET)*(1)/((automatika.cas));
			automatika.x_desired[4]	:= (automatika.x_desired_previous[4]*(automatika.cas - TIME_TO_INT(TON_0.ET))/automatika.cas) + TIME_TO_INT(TON_0.ET)*(1)/((automatika.cas));
			automatika.x_desired[5]	:= (automatika.x_desired_previous[5]*(automatika.cas - TIME_TO_INT(TON_0.ET))/automatika.cas) + TIME_TO_INT(TON_0.ET)*(1)/((automatika.cas));
			automatika.x_desired[6]	:= (automatika.x_desired_previous[6]*(automatika.cas - TIME_TO_INT(TON_0.ET))/automatika.cas) + TIME_TO_INT(TON_0.ET)*(1)/((automatika.cas));

			IF TON_0.Q = TRUE THEN
				automatika.casovac			:= FALSE;
				automatika.automatic		:= TRUE;
				global_step					:= 15;//12227
			END_IF

		12227:
			automatika.cas					:= 6000;
			global_step						:= 12228;
			FOR i:=0 TO 6 BY 1 DO
				automatika.x_desired_previous[i]:= automatika.x_desired[i];
				automatika.y_desired_previous[i]:= automatika.y_desired[i];
			END_FOR
			automatika.casovac				:= TRUE;

		12228:
			(*
			automatika.y_desired[0]	:= (automatika.y_desired_previous[0]*(automatika.cas - TIME_TO_INT(TON_0.ET))/automatika.cas) + TIME_TO_INT(TON_0.ET)*(REAL_TO_INT(packetPos.qDesired[0]))/((automatika.cas));
			automatika.y_desired[1]	:= (automatika.y_desired_previous[1]*(automatika.cas - TIME_TO_INT(TON_0.ET))/automatika.cas) + TIME_TO_INT(TON_0.ET)*(REAL_TO_INT(packetPos.qDesired[2]))/((automatika.cas));
			automatika.y_desired[2]	:= (automatika.y_desired_previous[2]*(automatika.cas - TIME_TO_INT(TON_0.ET))/automatika.cas) + TIME_TO_INT(TON_0.ET)*(REAL_TO_INT(packetPos.qDesired[4]))/((automatika.cas));
			automatika.y_desired[3]	:= (automatika.y_desired_previous[3]*(automatika.cas - TIME_TO_INT(TON_0.ET))/automatika.cas) + TIME_TO_INT(TON_0.ET)*(REAL_TO_INT(packetPos.qDesired[6]))/((automatika.cas));
			automatika.y_desired[4]	:= (automatika.y_desired_previous[4]*(automatika.cas - TIME_TO_INT(TON_0.ET))/automatika.cas) + TIME_TO_INT(TON_0.ET)*(REAL_TO_INT(packetPos.qDesired[8]))/((automatika.cas));
			automatika.y_desired[5]	:= (automatika.y_desired_previous[5]*(automatika.cas - TIME_TO_INT(TON_0.ET))/automatika.cas) + TIME_TO_INT(TON_0.ET)*(REAL_TO_INT(packetPos.qDesired[10]))/((automatika.cas));
			automatika.y_desired[6]	:= (automatika.y_desired_previous[6]*(automatika.cas - TIME_TO_INT(TON_0.ET))/automatika.cas) + TIME_TO_INT(TON_0.ET)*(REAL_TO_INT(packetPos.qDesired[12]))/((automatika.cas));

			automatika.x_desired[0]	:= (automatika.x_desired_previous[0]*(automatika.cas - TIME_TO_INT(TON_0.ET))/automatika.cas) + TIME_TO_INT(TON_0.ET)*(REAL_TO_INT(packetPos.qDesired[1]))/((automatika.cas));
			automatika.x_desired[1]	:= (automatika.x_desired_previous[1]*(automatika.cas - TIME_TO_INT(TON_0.ET))/automatika.cas) + TIME_TO_INT(TON_0.ET)*(REAL_TO_INT(packetPos.qDesired[3]))/((automatika.cas));
			automatika.x_desired[2]	:= (automatika.x_desired_previous[2]*(automatika.cas - TIME_TO_INT(TON_0.ET))/automatika.cas) + TIME_TO_INT(TON_0.ET)*(REAL_TO_INT(packetPos.qDesired[5]))/((automatika.cas));
			automatika.x_desired[3]	:= (automatika.x_desired_previous[3]*(automatika.cas - TIME_TO_INT(TON_0.ET))/automatika.cas) + TIME_TO_INT(TON_0.ET)*(REAL_TO_INT(packetPos.qDesired[7]))/((automatika.cas));
			automatika.x_desired[4]	:= (automatika.x_desired_previous[4]*(automatika.cas - TIME_TO_INT(TON_0.ET))/automatika.cas) + TIME_TO_INT(TON_0.ET)*(REAL_TO_INT(packetPos.qDesired[9]))/((automatika.cas));
			automatika.x_desired[5]	:= (automatika.x_desired_previous[5]*(automatika.cas - TIME_TO_INT(TON_0.ET))/automatika.cas) + TIME_TO_INT(TON_0.ET)*(REAL_TO_INT(packetPos.qDesired[11]))/((automatika.cas));
			automatika.x_desired[6]	:= (automatika.x_desired_previous[6]*(automatika.cas - TIME_TO_INT(TON_0.ET))/automatika.cas) + TIME_TO_INT(TON_0.ET)*(REAL_TO_INT(packetPos.qDesired[13]))/((automatika.cas));
			*)
			automatika.y_desired[0]	:= TIME_TO_INT(TON_0.ET)*(REAL_TO_INT(packetPos.qDesired[0]))/((automatika.cas));
			automatika.y_desired[1]	:= TIME_TO_INT(TON_0.ET)*(REAL_TO_INT(packetPos.qDesired[2]))/((automatika.cas));
			automatika.y_desired[2]	:= TIME_TO_INT(TON_0.ET)*(REAL_TO_INT(packetPos.qDesired[4]))/((automatika.cas));
			automatika.y_desired[3]	:= TIME_TO_INT(TON_0.ET)*(REAL_TO_INT(packetPos.qDesired[6]))/((automatika.cas));
			automatika.y_desired[4]	:= TIME_TO_INT(TON_0.ET)*(REAL_TO_INT(packetPos.qDesired[8]))/((automatika.cas));
			automatika.y_desired[5]	:= TIME_TO_INT(TON_0.ET)*(REAL_TO_INT(packetPos.qDesired[10]))/((automatika.cas));
			automatika.y_desired[6]	:= TIME_TO_INT(TON_0.ET)*(REAL_TO_INT(packetPos.qDesired[12]))/((automatika.cas));

			automatika.x_desired[0]	:= TIME_TO_INT(TON_0.ET)*(REAL_TO_INT(packetPos.qDesired[1]))/((automatika.cas));
			automatika.x_desired[1]	:= TIME_TO_INT(TON_0.ET)*(REAL_TO_INT(packetPos.qDesired[3]))/((automatika.cas));
			automatika.x_desired[2]	:= TIME_TO_INT(TON_0.ET)*(REAL_TO_INT(packetPos.qDesired[5]))/((automatika.cas));
			automatika.x_desired[3]	:= TIME_TO_INT(TON_0.ET)*(REAL_TO_INT(packetPos.qDesired[7]))/((automatika.cas));
			automatika.x_desired[4]	:= TIME_TO_INT(TON_0.ET)*(REAL_TO_INT(packetPos.qDesired[9]))/((automatika.cas));
			automatika.x_desired[5]	:= TIME_TO_INT(TON_0.ET)*(REAL_TO_INT(packetPos.qDesired[11]))/((automatika.cas));
			automatika.x_desired[6]	:= TIME_TO_INT(TON_0.ET)*(REAL_TO_INT(packetPos.qDesired[13]))/((automatika.cas));

			IF TON_0.Q THEN
				automatika.casovac				:= FALSE;
				FOR i:=0 TO 6 BY 1 DO
					automatika.I_konstanta[i]	:= 20;
				END_FOR
				automatika.automatic			:= TRUE;
				automatika.holdPosition			:= FALSE;
				global_step						:= 15;
				automatika.popcorn				:= FALSE;
			END_IF

		13:
			IF global_step_udp = 1 THEN
				automatika.effector			:= FALSE;
				//automatika.casovac_uchopenie:= TRUE;
				global_step					:= 14;
			END_IF

		14:
			//IF TON_1.Q = TRUE THEN
				automatika.casovac_uchopenie:= FALSE;
				global_step					:= 15;
			//END_IF

		15:
			IF global_step_udp = 2 THEN
				automatika.holdPosition		:= TRUE;
				automatika.cas				:= 1000;
				automatika.casovac			:= TRUE;
				global_step					:= 16;
			END_IF
		16:
			IF TON_0.Q = TRUE THEN
				automatika.casovac			:= FALSE;
				global_step					:= 17;
				automatika.popcorn			:= FALSE;
			END_IF
		17:	// pustenie objektu a cakanie na povel pokracovat
			IF global_step_udp = 3 THEN
				automatika.effector			:= FALSE;
				global_step					:= 18;
			END_IF

		18:
			IF global_step_udp = 4 THEN

				automatika.automatic		:= FALSE;
				automatika.holdPosition		:= FALSE;
				I_ON						:= FALSE;
				global_step					:= 19;//19
			END_IF

		19:

			FOR i:=0 TO 6 BY 1 DO
				automatika.x_desired_previous[i]	:= REAL_TO_INT(packetPos.qDesired[i*2]); //automatika.x_desired[i];
				automatika.y_desired_previous[i]	:= REAL_TO_INT(-packetPos.qDesired[i*2+1]); //automatika.y_desired[i];
				automatika.x_desired[i]				:= 0;
				automatika.y_desired[i]				:= 0;
				packetPos.qDesired[i*2]				:= 0;
				packetPos.qDesired[i*2+1]			:= 0;
				automatika.I_konstanta[i]			:= 5;
			END_FOR

			global_step				:= 20;
		20:
			I_ON					:= TRUE;
			automatika.cas			:= 5000;
			automatika.casovac		:= TRUE;
			global_step				:= 21;
		21:

			automatika.y_desired[0]	:= 0;
			automatika.y_desired[1]	:= 0;	// 5000ms
			automatika.y_desired[2]	:= 0;
			automatika.y_desired[3]	:= 0;
			automatika.y_desired[4]	:= 0;
			automatika.y_desired[5]	:= 0;
			automatika.y_desired[6]	:= 0;

			automatika.x_desired[0]	:= 0;
			automatika.x_desired[1]	:= 0;
			automatika.x_desired[2]	:= 0;
			automatika.x_desired[3]	:= 0;
			automatika.x_desired[4]	:= 0;
			automatika.x_desired[5]	:= 0;
			automatika.x_desired[6]	:= 0;
			(*
			automatika.y_desired[0]	:= (automatika.y_desired_previous[0]*(automatika.cas - TIME_TO_INT(TON_0.ET))/automatika.cas) + TIME_TO_INT(TON_0.ET)*(REAL_TO_INT(packetPos.qDesired[0]))/((automatika.cas));
			automatika.y_desired[1]	:= (automatika.y_desired_previous[1]*(automatika.cas - TIME_TO_INT(TON_0.ET))/automatika.cas) + TIME_TO_INT(TON_0.ET)*(REAL_TO_INT(packetPos.qDesired[0]))/((automatika.cas));
			automatika.y_desired[2]	:= (automatika.y_desired_previous[2]*(automatika.cas - TIME_TO_INT(TON_0.ET))/automatika.cas) + TIME_TO_INT(TON_0.ET)*(REAL_TO_INT(packetPos.qDesired[0]))/((automatika.cas));
			automatika.y_desired[3]	:= (automatika.y_desired_previous[3]*(automatika.cas - TIME_TO_INT(TON_0.ET))/automatika.cas) + TIME_TO_INT(TON_0.ET)*(REAL_TO_INT(packetPos.qDesired[0]))/((automatika.cas));
			automatika.y_desired[4]	:= (automatika.y_desired_previous[4]*(automatika.cas - TIME_TO_INT(TON_0.ET))/automatika.cas) + TIME_TO_INT(TON_0.ET)*(REAL_TO_INT(packetPos.qDesired[0]))/((automatika.cas));
			automatika.y_desired[5]	:= (automatika.y_desired_previous[5]*(automatika.cas - TIME_TO_INT(TON_0.ET))/automatika.cas) + TIME_TO_INT(TON_0.ET)*(REAL_TO_INT(packetPos.qDesired[0]))/((automatika.cas));
			automatika.y_desired[6]	:= (automatika.y_desired_previous[6]*(automatika.cas - TIME_TO_INT(TON_0.ET))/automatika.cas) + TIME_TO_INT(TON_0.ET)*(REAL_TO_INT(packetPos.qDesired[0]))/((automatika.cas));

			automatika.x_desired[0]	:= (automatika.x_desired_previous[0]*(automatika.cas - TIME_TO_INT(TON_0.ET))/automatika.cas) + TIME_TO_INT(TON_0.ET)*(REAL_TO_INT(packetPos.qDesired[1]))/((automatika.cas));
			automatika.x_desired[1]	:= (automatika.x_desired_previous[1]*(automatika.cas - TIME_TO_INT(TON_0.ET))/automatika.cas) + TIME_TO_INT(TON_0.ET)*(REAL_TO_INT(packetPos.qDesired[1]))/((automatika.cas));
			automatika.x_desired[2]	:= (automatika.x_desired_previous[2]*(automatika.cas - TIME_TO_INT(TON_0.ET))/automatika.cas) + TIME_TO_INT(TON_0.ET)*(REAL_TO_INT(packetPos.qDesired[1]))/((automatika.cas));
			automatika.x_desired[3]	:= (automatika.x_desired_previous[3]*(automatika.cas - TIME_TO_INT(TON_0.ET))/automatika.cas) + TIME_TO_INT(TON_0.ET)*(REAL_TO_INT(packetPos.qDesired[1]))/((automatika.cas));
			automatika.x_desired[4]	:= (automatika.x_desired_previous[4]*(automatika.cas - TIME_TO_INT(TON_0.ET))/automatika.cas) + TIME_TO_INT(TON_0.ET)*(REAL_TO_INT(packetPos.qDesired[1]))/((automatika.cas));
			automatika.x_desired[5]	:= (automatika.x_desired_previous[5]*(automatika.cas - TIME_TO_INT(TON_0.ET))/automatika.cas) + TIME_TO_INT(TON_0.ET)*(REAL_TO_INT(packetPos.qDesired[1]))/((automatika.cas));
			automatika.x_desired[6]	:= (automatika.x_desired_previous[6]*(automatika.cas - TIME_TO_INT(TON_0.ET))/automatika.cas) + TIME_TO_INT(TON_0.ET)*(REAL_TO_INT(packetPos.qDesired[1]))/((automatika.cas));
			*)
			automatika.linear		:= 23;

			IF TON_0.Q = TRUE THEN
				automatika.casovac	:= FALSE;
				global_step			:= 999;
			END_IF

			(*
			FOR i:=0 TO 6 BY 1 DO
				packetPos.qDesired[i*2]		:= 0;
				packetPos.qDesired[i*2+1]	:= 0;
				automatika.y_desired[i]		:= 0;
				automatika.x_desired[i]		:= 0;
			END_FOR
		*)

		//	IF TON_0.Q = TRUE THEN
		//		automatika.casovac		:= FALSE;
				//	global_step				:= 999;
		//	END_IF

		//	global_step						:= 20;

		22:

			(*
			automatika.y_desired[0]	:= TIME_TO_INT(TON_0.ET)*(1)/((automatika.cas));
			automatika.y_desired[1]	:= TIME_TO_INT(TON_0.ET)*(1)/((automatika.cas));	// 5000ms
			automatika.y_desired[2]	:= TIME_TO_INT(TON_0.ET)*(1)/((automatika.cas));
			automatika.y_desired[3]	:= TIME_TO_INT(TON_0.ET)*(1)/((automatika.cas));
			automatika.y_desired[4]	:= TIME_TO_INT(TON_0.ET)*(1)/((automatika.cas));
			automatika.y_desired[5]	:= TIME_TO_INT(TON_0.ET)*(1)/((automatika.cas));
			automatika.y_desired[6]	:= TIME_TO_INT(TON_0.ET)*(1)/((automatika.cas));

			automatika.x_desired[0]	:= TIME_TO_INT(TON_0.ET)*(1)/((automatika.cas));
			automatika.x_desired[1]	:= TIME_TO_INT(TON_0.ET)*(1)/((automatika.cas));
			automatika.x_desired[2]	:= TIME_TO_INT(TON_0.ET)*(1)/((automatika.cas));
			automatika.x_desired[3]	:= TIME_TO_INT(TON_0.ET)*(1)/((automatika.cas));
			automatika.x_desired[4]	:= TIME_TO_INT(TON_0.ET)*(1)/((automatika.cas));
			automatika.x_desired[5]	:= TIME_TO_INT(TON_0.ET)*(1)/((automatika.cas));
			*)
			(*
			automatika.y_desired[0]	:= (automatika.y_desired_previous[0]*(automatika.cas - TIME_TO_INT(TON_0.ET))/automatika.cas) + TIME_TO_INT(TON_0.ET)*(1)/((automatika.cas));
			automatika.y_desired[1]	:= (automatika.y_desired_previous[1]*(automatika.cas - TIME_TO_INT(TON_0.ET))/automatika.cas) + TIME_TO_INT(TON_0.ET)*(1)/((automatika.cas));	// 5000ms
			automatika.y_desired[2]	:= (automatika.y_desired_previous[2]*(automatika.cas - TIME_TO_INT(TON_0.ET))/automatika.cas) + TIME_TO_INT(TON_0.ET)*(1)/((automatika.cas));
			automatika.y_desired[3]	:= (automatika.y_desired_previous[3]*(automatika.cas - TIME_TO_INT(TON_0.ET))/automatika.cas) + TIME_TO_INT(TON_0.ET)*(1)/((automatika.cas));
			automatika.y_desired[4]	:= (automatika.y_desired_previous[4]*(automatika.cas - TIME_TO_INT(TON_0.ET))/automatika.cas) + TIME_TO_INT(TON_0.ET)*(1)/((automatika.cas));
			automatika.y_desired[5]	:= (automatika.y_desired_previous[5]*(automatika.cas - TIME_TO_INT(TON_0.ET))/automatika.cas) + TIME_TO_INT(TON_0.ET)*(1)/((automatika.cas));
			automatika.y_desired[6]	:= (automatika.y_desired_previous[6]*(automatika.cas - TIME_TO_INT(TON_0.ET))/automatika.cas) + TIME_TO_INT(TON_0.ET)*(1)/((automatika.cas));

			automatika.x_desired[0]	:= (automatika.x_desired_previous[0]*(automatika.cas - TIME_TO_INT(TON_0.ET))/automatika.cas) + TIME_TO_INT(TON_0.ET)*(1)/((automatika.cas));
			automatika.x_desired[1]	:= (automatika.x_desired_previous[1]*(automatika.cas - TIME_TO_INT(TON_0.ET))/automatika.cas) + TIME_TO_INT(TON_0.ET)*(1)/((automatika.cas));
			automatika.x_desired[2]	:= (automatika.x_desired_previous[2]*(automatika.cas - TIME_TO_INT(TON_0.ET))/automatika.cas) + TIME_TO_INT(TON_0.ET)*(1)/((automatika.cas));
			automatika.x_desired[3]	:= (automatika.x_desired_previous[3]*(automatika.cas - TIME_TO_INT(TON_0.ET))/automatika.cas) + TIME_TO_INT(TON_0.ET)*(1)/((automatika.cas));
			automatika.x_desired[4]	:= (automatika.x_desired_previous[4]*(automatika.cas - TIME_TO_INT(TON_0.ET))/automatika.cas) + TIME_TO_INT(TON_0.ET)*(1)/((automatika.cas));
			automatika.x_desired[5]	:= (automatika.x_desired_previous[5]*(automatika.cas - TIME_TO_INT(TON_0.ET))/automatika.cas) + TIME_TO_INT(TON_0.ET)*(1)/((automatika.cas));
			automatika.x_desired[6]	:= (automatika.x_desired_previous[6]*(automatika.cas - TIME_TO_INT(TON_0.ET))/automatika.cas) + TIME_TO_INT(TON_0.ET)*(1)/((automatika.cas));
			*)

	END_CASE

END_PROGRAM
```

### Program Logical/Source/UDP/Client (IEC) - AsUDP Client Application

#### Client.st - Cyclic code
```iecst
(********************************************************************
 * COPYRIGHT -- Bernecker + Rainer
 ********************************************************************
 * Program: Client
 * File: Client.st
 * Author: Bernecker + Rainer
 * Created: June 02, 2008
 ********************************************************************
 * Implementation of program Client
 ********************************************************************)

PROGRAM _CYCLIC

	//LibAsUDP1_ST.send_data[0] := LibAsUDP1_ST.send_data[0] + 1;  (* Generate a "running" variable for Data transfer *)
	//LibAsUDP1_ST.send_data := '20.12 12.54 10.24 -13.25';
	(*
	memset(ADR(LibAsUDP1_ST.send_data), 0, SIZEOF(LibAsUDP1_ST.send_data));
	memset(ADR(helpString), 0, SIZEOF(helpString));

	FOR i:=0 TO 6 BY 1 DO
		ftoa(modul.uhol_XminusRef[i], ADR(helpString));
		strcat(ADR(LibAsUDP1_ST.send_data), ADR(helpString));
		strcat(ADR(LibAsUDP1_ST.send_data), ADR(','));
		ftoa(modul.uhol_YminusRef[i], ADR(helpString));
		strcat(ADR(LibAsUDP1_ST.send_data), ADR(helpString));
		strcat(ADR(LibAsUDP1_ST.send_data), ADR(','));
	END_FOR
	ftoa(modul.linearReal, ADR(helpString)); // vymenit za linearny
	strcat(ADR(LibAsUDP1_ST.send_data), ADR(helpString));
	*)
	//strcat(ADR(LibAsUDP1_ST.send_data), ADR(','));

	memset(ADR(LibAsUDP1_ST.send_data), 0, SIZEOF(LibAsUDP1_ST.send_data));
	IF (automatika.step_repeatability=44) OR (automatika.step_repeatability=77) OR (automatika.step_repeatability=99) THEN
		strcat(ADR(LibAsUDP1_ST.send_data), ADR('1'));
	ELSE
		strcat(ADR(LibAsUDP1_ST.send_data), ADR('0'));
	END_IF

	(*
	memset(ADR(LibAsUDP1_ST.send_data), 0, SIZEOF(LibAsUDP1_ST.send_data));
	memset(ADR(helpString), 0, SIZEOF(helpString));

	FOR i:=0 TO 5 BY 1 DO
		ftoa(modul.uhol1[i], ADR(helpString));
		strcat(ADR(LibAsUDP1_ST.send_data), ADR(helpString));
		strcat(ADR(LibAsUDP1_ST.send_data), ADR(','));
		ftoa(modul.uhol2[i], ADR(helpString));
		strcat(ADR(LibAsUDP1_ST.send_data), ADR(helpString));
		strcat(ADR(LibAsUDP1_ST.send_data), ADR(','));
	END_FOR
	ftoa(modul.uhol2[0], ADR(helpString)); // vymenit za linearny
	strcat(ADR(LibAsUDP1_ST.send_data), ADR(helpString));
	//strcat(ADR(LibAsUDP1_ST.send_data), ADR(','));
	*)
	CASE Client.sStep OF

		0:	(* Open UDP Port *)
			Client.UdpOpen_0.enable := 1;
			Client.UdpOpen_0.pIfAddr := 0;	(* Listen on all TCP/IP Interfaces*)
			Client.UdpOpen_0.port := 12051;	(* Port to listen*)
			Client.UdpOpen_0.options := 0;
			Client.UdpOpen_0;	(* Call the Function*)

			IF Client.UdpOpen_0.status = 0 THEN  (* UdpOpen successful*)
				Client.sStep := 1;
			ELSIF Client.UdpOpen_0.status = ERR_FUB_BUSY THEN  (* UdpOpen not finished -> redo *)
			  (* Busy *)
			ELSE  (* Goto Error Step *)
				Client.sStep := 10;
			END_IF

		1:	(* Send Data to the Server *)
			Client.server_address := '192.168.1.47';	(* IP Address of the Server *)
			Client.server_portnumber := 12050;	(* Port number of the Server *)

			Client.UdpSend_0.enable := 1;
			Client.UdpSend_0.ident := Client.UdpOpen_0.ident;	(* Connection Ident from AsUDP.UDP_Open *)
			Client.UdpSend_0.pHost := ADR(Client.server_address);
			Client.UdpSend_0.port := Client.server_portnumber;
			Client.UdpSend_0.pData := ADR(LibAsUDP1_ST.send_data);	(* Which data to send *)
			Client.UdpSend_0.datalen := SIZEOF(LibAsUDP1_ST.send_data);	(* Lenght of data to send *)
			Client.UdpSend_0.flags := 0;
			Client.UdpSend_0;	(* Call the Function*)

			IF Client.UdpSend_0.status = 0 THEN  (* Data sent *)
				Client.sStep := 2;
			ELSIF Client.UdpSend_0.status = ERR_FUB_BUSY THEN  (* UdpSend not finished -> redo *)
			  (* Busy *)
			ELSE  (* Goto Error Step *)
				Client.sStep := 10;
			END_IF

		2:	(* Receive Data from the Server *)
			Client.UdpRecv_0.enable := 1;
			Client.UdpRecv_0.ident := Client.UdpOpen_0.ident;  (* Connection Ident from AsUDP.UDP_Open *)
			Client.UdpRecv_0.pData	:= ADR(LibAsUDP1_ST.receive_data);  (* Where to store the incoming data *)//ADR(LibAsUDP1_ST.receive_data);
			Client.UdpRecv_0.datamax := SIZEOF(LibAsUDP1_ST.receive_data);  (* Lenght of data buffer *)
			Client.UdpRecv_0.flags := 0;
			Client.UdpRecv_0;  (* Call the Function*)

			IF Client.UdpRecv_0.status = 0 THEN  (* Data was received successfully -> Send next packet *)
				Client.sStep := 3;
				Client.no_data_received_count := 0;
			ELSIF Client.UdpRecv_0.status = udpERR_NO_DATA THEN  (* No data received - wait *)
			  (* No Data received *)
			  	Client.no_data_received_count := Client.no_data_received_count + 1;	(* Increase if no data are received *)

				IF Client.no_data_received_count > 200 THEN		(* No data timeout for TC1 [10ms] *)
					Client.no_data_received_count := 0;
					Client.sStep := 1;	(* Send again *)
				END_IF
			ELSIF Client.UdpRecv_0.status = ERR_FUB_BUSY THEN  (* UdpRecv not finished -> redo *)
			  (* Busy *)
			ELSE  (* Goto Error Step *)
				Client.sStep := 10;
			END_IF

		3: (* Close connection *)
			Client.UdpClose_0.enable := 1;
			Client.UdpClose_0.ident := Client.UdpOpen_0.ident;  (* Connection Ident from AsUDP.UDP_Open *)
			Client.UdpClose_0;  (* Call the Function*)

			IF Client.UdpClose_0.status = 0 THEN  (* Close successful -> Reopen the interface *)
				Client.sStep := 0;
			ELSIF Client.UdpClose_0.status = ERR_FUB_BUSY THEN  (* UdpClose not finished -> redo *)
			  (* Busy *)
			ELSE  (* Goto Error Step *)
				Client.sStep := 10;
			END_IF

		10: (* Here some error Handling has to be implemented *)

	END_CASE

END_PROGRAM
```

#### Client.typ - UDP Client Variables
```iecst
(********************************************************************
 * COPYRIGHT -- Bernecker + Rainer
 ********************************************************************
 * Program: Client
 * File: Client.typ
 * Author: Bernecker + Rainer
 * Created: June 02, 2008
 ********************************************************************
 * Local data types of program Client
 ********************************************************************)

TYPE
	Client_typ : 	STRUCT  (*UDP Client Variables*)
		sStep : UINT; (*UDP Client Step Variable*)
		server_address : STRING[20]; (*Address of the Server*)
		server_portnumber : UINT; (*Portnumber of the Server*)
		no_data_received_count : UINT; (*Counts up if no data are received*)
		UdpOpen_0 : UdpOpen; (*AsUDP.UdpOpen FUB*)
		UdpConnect_0 : UdpConnect; (*AsUDP.UdpConnect FUB*)
		UdpSend_0 : UdpSend; (*AsUDP.UdpSend FUB*)
		UdpRecv_0 : UdpRecv; (*AsUDP.UdpRecv FUB*)
		UdpDisconnect_0 : UdpDisconnect; (*AsUDP.UdpDisconnect FUB*)
		UdpClose_0 : UdpClose; (*AsUDP.UdpClose FUB*)
	END_STRUCT;
END_TYPE
```

### Program Logical/Source/Controller (IEC)

#### Variables.var
```iecst
VAR
	Vin_x_prechodne : REAL;
	Vin_y_prechodne : REAL;
	pocitadlo : INT;
	Vin_x_priemer : REAL;
	Vin_y_priemer : REAL;
	cos_test : BOOL;
	kalibracia_x : REAL;
	kalibracia_y : REAL;
	uhol_y_predosly : REAL;
	uhol_x_predosly : REAL;
	pozadovany_uhol_y_predosly : REAL;
	x1 : REAL := 5;
	y1 : REAL := 75;
	x2 : REAL := 1;
	y2 : REAL := 350;
	a : REAL;
	b : REAL;
	error_x : REAL;
	error_total : REAL;
	error_y : REAL;
	modull : mech;
	test_const_I : BOOL := FALSE;
	pozadovany_uhol_x_predosly : REAL;
	p11 : REAL;
	p22 : REAL;
	p33 : REAL;
	stlacene : BOOL;
	poradie : INT;
	pozadovany_uhol_x_old : REAL;
	pozadovany_uhol_y_old : REAL;
	i : INT;
	FF_PID_r_t_3 : FF_PID_r_t;
	FF_PID_r_t_0 : FF_PID_r_t;
	id : INT;
	FF_PID_r_t_1 : FF_PID_r_t;
	FF_PID_r_t_2 : FF_PID_r_t;
	I_ON : BOOL;
	switch : BOOL;
	maxUhol : INT;
	TON_0 : TON;
	kalibraciaStart : BOOL;
	TON_1 : TON;
	switch2 : BOOL;
END_VAR
```
